	{attribute 'TcIecLibraryType'}
	{attribute 'external_name' := 'F_VN_ImageAbsoluteAverage_GUID_2A28D3C0_C84C_D0B6_A685_B52828B14CE3'}
	(* Computes the average absolute pixel value of an image. *)
	FUNCTION F_VN_ImageAbsoluteAverage : HRESULT
	VAR_INPUT
		ipSrcImage	:	ITcVnImage;	(* Source image *)
	END_VAR
	VAR_IN_OUT
		fAverage	:	LREAL;	(* Returns the average absolute pixel value *)
	END_VAR
	VAR_INPUT
		hrPrev	:	HRESULT;	(* HRESULT indicating the result of previous operations (If SUCCEEDED(hrPrev) equals false, no operation is executed.) *)
	END_VAR

END_FUNCTION

// Functions/Image Analysis/F_VN_ImageAverage

	{attribute 'TcIecLibraryType'}
	{attribute 'external_name' := 'F_VN_ImageAverage_GUID_FE774972_76AD_D27D_BAED_5933ADCB3F82'}
	(* Computes the (channel-wise) average pixel value of an image. *)
	FUNCTION F_VN_ImageAverage : HRESULT
	VAR_INPUT
		ipSrcImage	:	ITcVnImage;	(* Source image (1 - 4 channels) *)
	END_VAR
	VAR_IN_OUT
		aAverage	:	TcVnVector4_LREAL;	(* Returns the (channel-wise) average pixel value of ipSrcImage *)
	END_VAR
	VAR_INPUT
		hrPrev	:	HRESULT;	(* HRESULT indicating the result of previous operations (If SUCCEEDED(hrPrev) equals false, no operation is executed.) *)
	END_VAR

END_FUNCTION

// Functions/Image Analysis/F_VN_ImageAverageExp

	{attribute 'TcIecLibraryType'}
	{attribute 'external_name' := 'F_VN_ImageAverageExp_GUID_3E21A3C6_8FFA_DAD8_9B62_448D6BE9A6F9'}
	(* Computes the (channel-wise) average pixel value of an image. (expert function) *)
	FUNCTION F_VN_ImageAverageExp : HRESULT
	VAR_INPUT
		ipSrcImage	:	ITcVnImage;	(* Source image (1 - 4 channels) *)
	END_VAR
	VAR_IN_OUT
		aAverage	:	TcVnVector4_LREAL;	(* Returns the (channel-wise) average pixel value of ipSrcImage *)
	END_VAR
	VAR_INPUT
		ipMask	:	ITcVnImage;	(* Mask of type USINT (1 channel) *)
		hrPrev	:	HRESULT;	(* HRESULT indicating the result of previous operations (If SUCCEEDED(hrPrev) equals false, no operation is executed.) *)
	END_VAR

END_FUNCTION

// Functions/Image Analysis/F_VN_ImageAverageStdDev

	{attribute 'TcIecLibraryType'}
	{attribute 'external_name' := 'F_VN_ImageAverageStdDev_GUID_C9B349AB_3E58_D491_BF33_2DB560BD56B6'}
	(* Computes the (channel-wise) average pixel value and the corresponding standard deviation of an image. *)
	FUNCTION F_VN_ImageAverageStdDev : HRESULT
	VAR_INPUT
		ipSrcImage	:	ITcVnImage;	(* Source image (1 - 4 channels) *)
	END_VAR
	VAR_IN_OUT
		aAverage	:	TcVnVector4_LREAL;	(* Returns the (channel-wise) average pixel value of ipSrcImage *)
		aStdDev	:	TcVnVector4_LREAL;	(* Returns the (channel-wise) pixel value standard deviation of ipSrcImage *)
	END_VAR
	VAR_INPUT
		hrPrev	:	HRESULT;	(* HRESULT indicating the result of previous operations (If SUCCEEDED(hrPrev) equals false, no operation is executed.) *)
	END_VAR

END_FUNCTION

// Functions/Image Analysis/F_VN_ImageAverageStdDevExp

	{attribute 'TcIecLibraryType'}
	{attribute 'external_name' := 'F_VN_ImageAverageStdDevExp_GUID_869E8E6A_9652_D404_9B63_9DC2492C3981'}
	(* Computes the (channel-wise) average pixel value and the corresponding standard deviation of an image. (expert function) *)
	FUNCTION F_VN_ImageAverageStdDevExp : HRESULT
	VAR_INPUT
		ipSrcImage	:	ITcVnImage;	(* Source image (1 - 4 channels) *)
	END_VAR
	VAR_IN_OUT
		aAverage	:	TcVnVector4_LREAL;	(* Returns the (channel-wise) average pixel value of ipSrcImage *)
		aStdDev	:	TcVnVector4_LREAL;	(* Returns the (channel-wise) pixel value standard deviation of ipSrcImage *)
	END_VAR
	VAR_INPUT
		ipMask	:	ITcVnImage;	(* Mask of type USINT (1 channel) *)
		hrPrev	:	HRESULT;	(* HRESULT indicating the result of previous operations (If SUCCEEDED(hrPrev) equals false, no operation is executed.) *)
	END_VAR

END_FUNCTION

// Functions/Image Analysis/F_VN_ImageCenterOfMass

	{attribute 'TcIecLibraryType'}
	{attribute 'external_name' := 'F_VN_ImageCenterOfMass_GUID_E26AB96A_EBBA_D4BE_88C4_CC4D119BCFE3'}
	(* Computes the center of mass of an image. *)
	FUNCTION F_VN_ImageCenterOfMass : HRESULT
	VAR_INPUT
		ipSrcImage	:	ITcVnImage;	(* Source image (1 channel) *)
	END_VAR
	VAR_IN_OUT
		aCenterOfMass	:	TcVnPoint2_LREAL;	(* Returns the center of mass of the image *)
	END_VAR
	VAR_INPUT
		hrPrev	:	HRESULT;	(* HRESULT indicating the result of previous operations (If SUCCEEDED(hrPrev) equals false, no operation is executed.) *)
	END_VAR

END_FUNCTION

// Functions/Image Analysis/F_VN_ImageCenterOfMassExp

	{attribute 'TcIecLibraryType'}
	{attribute 'external_name' := 'F_VN_ImageCenterOfMassExp_GUID_59EB1D9F_B0E1_D491_9AD3_AE15A5EDCA0C'}
	(* Computes the center of mass of an image. *)
	FUNCTION F_VN_ImageCenterOfMassExp : HRESULT
	VAR_INPUT
		ipSrcImage	:	ITcVnImage;	(* Source image (1 channel) *)
	END_VAR
	VAR_IN_OUT
		aCenterOfMass	:	TcVnPoint2_LREAL;	(* Returns the center of mass of the image *)
	END_VAR
	VAR_INPUT
		ipMask	:	ITcVnImage;	(* Optional mask (1 channel of type USINT, same width and height as ipSrcImage) *)
		hrPrev	:	HRESULT;	(* HRESULT indicating the result of previous operations (If SUCCEEDED(hrPrev) equals false, no operation is executed.) *)
	END_VAR

END_FUNCTION

// Functions/Image Analysis/F_VN_ImageMedian

	{attribute 'TcIecLibraryType'}
	{attribute 'external_name' := 'F_VN_ImageMedian_GUID_F4FC4EAF_2294_D8BC_B4E8_1BD025C52AE2'}
	(* Computes the (approximated, channel-wise) median pixel value of an image. *)
	FUNCTION F_VN_ImageMedian : HRESULT
	VAR_INPUT
		ipSrcImage	:	ITcVnImage;	(* Source image (1 - 4 channels) *)
	END_VAR
	VAR_IN_OUT
		aMedian	:	TcVnVector4_LREAL;	(* Returns the (approximated, channel-wise) median pixel value of ipSrcImage *)
	END_VAR
	VAR_INPUT
		hrPrev	:	HRESULT;	(* HRESULT indicating the result of previous operations (If SUCCEEDED(hrPrev) equals false, no operation is executed.) *)
	END_VAR

END_FUNCTION

// Functions/Image Analysis/F_VN_ImageMedianExp

	{attribute 'TcIecLibraryType'}
	{attribute 'external_name' := 'F_VN_ImageMedianExp_GUID_743A193B_E592_DD8C_9D14_320E1F951A29'}
	(* Computes the (approximated, channel-wise) median pixel value of an image. (expert function) *)
	FUNCTION F_VN_ImageMedianExp : HRESULT
	VAR_INPUT
		ipSrcImage	:	ITcVnImage;	(* Source image (1 - 4 channels) *)
	END_VAR
	VAR_IN_OUT
		aMedian	:	TcVnVector4_LREAL;	(* Returns the (approximated, channel-wise) median pixel value of ipSrcImage *)
	END_VAR
	VAR_INPUT
		ipMask	:	ITcVnImage;	(* Mask of type USINT (1 channel) *)
		hrPrev	:	HRESULT;	(* HRESULT indicating the result of previous operations (If SUCCEEDED(hrPrev) equals false, no operation is executed.) *)
	END_VAR

END_FUNCTION

// Functions/Image Analysis/F_VN_ImageMoments

	{attribute 'TcIecLibraryType'}
	{attribute 'external_name' := 'F_VN_ImageMoments_GUID_E6E09E69_C28D_D19A_BF53_C7F25960A9B6'}
	(* Computes the spatial moments, the central moments, and the central normalized moments of an image up to the third order. *)
	FUNCTION F_VN_ImageMoments : HRESULT
	VAR_INPUT
		ipImage	:	ITcVnImage;	(* Source image (1 channel, elements of type USINT or REAL) *)
	END_VAR
	VAR_IN_OUT
		stMoments	:	TcVnMoments;	(* Returns a struct containing the moments *)
	END_VAR
	VAR_INPUT
		bBinaryImage	:	BOOL;	(* If true, all non-zero pixels are treated as ones *)
		hrPrev	:	HRESULT;	(* HRESULT indicating the result of previous operations (If SUCCEEDED(hrPrev) equals false, no operation is executed.) *)
	END_VAR

END_FUNCTION

// Functions/Image Analysis/F_VN_MaxPixelValue

	{attribute 'TcIecLibraryType'}
	{attribute 'external_name' := 'F_VN_MaxPixelValue_GUID_31A56A5D_0E05_D01A_8DEF_0E54450C3D06'}
	(* Finds the maximum pixel value in an image (1 - 4 channels supported). *)
	FUNCTION F_VN_MaxPixelValue : HRESULT
	VAR_INPUT
		ipImage	:	ITcVnImage;	(* Source image *)
	END_VAR
	VAR_IN_OUT
		aMaxValue	:	TcVnVector4_LREAL;	(* Returns the maximum pixel value *)
		aPosition	:	TcVnPoint2_DINT;	(* Returns the first found position of aMaxValue *)
	END_VAR
	VAR_INPUT
		hrPrev	:	HRESULT;	(* HRESULT indicating the result of previous operations (If SUCCEEDED(hrPrev) equals false, no operation is executed.) *)
	END_VAR

END_FUNCTION

// Functions/Image Analysis/F_VN_MaxPixelValueExp

	{attribute 'TcIecLibraryType'}
	{attribute 'external_name' := 'F_VN_MaxPixelValueExp_GUID_1D7E82B6_8AF8_D9FA_862F_06A78D41E2CB'}
	(* Finds the maximum pixel value in an image (1 - 4 channels supported). (expert function) *)
	FUNCTION F_VN_MaxPixelValueExp : HRESULT
	VAR_INPUT
		ipImage	:	ITcVnImage;	(* Source image *)
	END_VAR
	VAR_IN_OUT
		aMaxValue	:	TcVnVector4_LREAL;	(* Returns the maximum pixel value *)
		aPosition	:	TcVnPoint2_DINT;	(* Returns the first found position of aMaxValue (not supported for multi-channel images with ELEMENTWISE) *)
	END_VAR
	VAR_INPUT
		ipMask	:	ITcVnImage;	(* Optional mask to specify which pixel positions are considered (USINT, set parameter to 0 if not required) *)
		eVectorCompareMethod	:	ETcVnVectorCompareMethod;	(* Select a vector compare method for multi-channel images *)
		hrPrev	:	HRESULT;	(* HRESULT indicating the result of previous operations (If SUCCEEDED(hrPrev) equals false, no operation is executed.) *)
	END_VAR

END_FUNCTION

// Functions/Image Analysis/F_VN_MinPixelValue

	{attribute 'TcIecLibraryType'}
	{attribute 'external_name' := 'F_VN_MinPixelValue_GUID_5C49F054_DDB2_D937_AA1E_11C3D82EEE93'}
	(* Finds the minimum pixel value in an image (1 - 4 channels supported). *)
	FUNCTION F_VN_MinPixelValue : HRESULT
	VAR_INPUT
		ipImage	:	ITcVnImage;	(* Source image *)
	END_VAR
	VAR_IN_OUT
		aMinValue	:	TcVnVector4_LREAL;	(* Returns the minimum pixel value *)
		aPosition	:	TcVnPoint2_DINT;	(* Returns the first found position of aMinValue *)
	END_VAR
	VAR_INPUT
		hrPrev	:	HRESULT;	(* HRESULT indicating the result of previous operations (If SUCCEEDED(hrPrev) equals false, no operation is executed.) *)
	END_VAR

END_FUNCTION

// Functions/Image Analysis/F_VN_MinPixelValueExp

	{attribute 'TcIecLibraryType'}
	{attribute 'external_name' := 'F_VN_MinPixelValueExp_GUID_843B3B42_9C53_D824_9E8C_EE174779F5B7'}
	(* Finds the minimum pixel value in an image (1 - 4 channels supported). (expert function) *)
	FUNCTION F_VN_MinPixelValueExp : HRESULT
	VAR_INPUT
		ipImage	:	ITcVnImage;	(* Source image *)
	END_VAR
	VAR_IN_OUT
		aMinValue	:	TcVnVector4_LREAL;	(* Returns the minimum pixel value *)
		aPosition	:	TcVnPoint2_DINT;	(* Returns the first found position of aMinValue (not supported for multi-channel images with ELEMENTWISE) *)
	END_VAR
	VAR_INPUT
		ipMask	:	ITcVnImage;	(* Optional mask to specify which pixel positions are considered (USINT, set parameter to 0 if not required) *)
		eVectorCompareMethod	:	ETcVnVectorCompareMethod;	(* Select a vector compare method for multi-channel images *)
		hrPrev	:	HRESULT;	(* HRESULT indicating the result of previous operations (If SUCCEEDED(hrPrev) equals false, no operation is executed.) *)
	END_VAR

END_FUNCTION

// Functions/Image Analysis/F_VN_RegionOrientation

	{attribute 'TcIecLibraryType'}
	{attribute 'external_name' := 'F_VN_RegionOrientation_GUID_3030DDA5_1563_D8A7_A605_14FE25F90FB6'}
	(* Calculate the orientation of a region based on a binary image that contains a non zero value for every pixel in that region. *)
	FUNCTION F_VN_RegionOrientation : HRESULT
	VAR_INPUT
		ipSrcImage	:	ITcVnImage;	(* Source image (1 channel, binary). *)
	END_VAR
	VAR_IN_OUT
		stOrientation	:	TcVnRotatedRectangle;	(* Resulting rotated rectangle, containig center of mass, lenghts of axes, and rotation angle of the region in clockwise direction. *)
	END_VAR
	VAR_INPUT
		hrPrev	:	HRESULT;	(* HRESULT indicating the result of previous operations (If SUCCEEDED(hrPrev) equals false, no operation is executed.) *)
	END_VAR

END_FUNCTION

// Functions/Image Analysis/F_VN_RegionOrientationExp

	{attribute 'TcIecLibraryType'}
	{attribute 'external_name' := 'F_VN_RegionOrientationExp_GUID_2D852B8B_71E3_D6E2_B2E4_953101B92198'}
	(* Calculate the orientation of a region based on a binary image that contains a non zero value for every pixel in that region. (expert function) *)
	FUNCTION F_VN_RegionOrientationExp : HRESULT
	VAR_INPUT
		ipSrcImage	:	ITcVnImage;	(* Source image (1 channel, binary) *)
	END_VAR
	VAR_IN_OUT
		stOrientation	:	TcVnRotatedRectangle;	(* Resulting rotated rectangle, containig center of mass, lenghts of axes, and rotation angle of the region in clockwise direction. *)
	END_VAR
	VAR_INPUT
		eMethod	:	ETcVnOrientationMethod;	(* Method for calculating the orientation. *)
		hrPrev	:	HRESULT;	(* HRESULT indicating the result of previous operations (If SUCCEEDED(hrPrev) equals false, no operation is executed.) *)
	END_VAR

END_FUNCTION

// Functions/Image Analysis/F_VN_UprightInnerRectangle

	{attribute 'TcIecLibraryType'}
	{attribute 'external_name' := 'F_VN_UprightInnerRectangle_GUID_9A6E9260_7D1F_D847_92B8_836A9953FD1A'}
	(* Computes the maximum area upright inner rectangle inside an area. If the valid area contains very small invalid areas or the performance is too slow, use the expert variant of this function and manually choose a suitable nDownScaleFactor. *)
	FUNCTION F_VN_UprightInnerRectangle : HRESULT
	VAR_INPUT
		ipSrcImage	:	ITcVnImage;	(* Source image (USINT, 1 channel, binary, values > 0 mark valid area) *)
	END_VAR
	VAR_IN_OUT
		stRectangle	:	TcVnRectangle_DINT;	(* Returns the maximum area upright inner rectangle *)
	END_VAR
	VAR_INPUT
		hrPrev	:	HRESULT;	(* HRESULT indicating the result of previous operations (If SUCCEEDED(hrPrev) equals false, no operation is executed.) *)
	END_VAR

END_FUNCTION

// Functions/Image Analysis/F_VN_UprightInnerRectangleExp

	{attribute 'TcIecLibraryType'}
	{attribute 'external_name' := 'F_VN_UprightInnerRectangleExp_GUID_86F2F7A8_492B_D31B_B473_8128A9E0833D'}
	(* Computes the maximum area upright inner rectangle inside an area. (expert function) *)
	FUNCTION F_VN_UprightInnerRectangleExp : HRESULT
	VAR_INPUT
		ipSrcImage	:	ITcVnImage;	(* Source image (USINT, 1 channel, binary, values > 0 mark valid area) *)
	END_VAR
	VAR_IN_OUT
		stRectangle	:	TcVnRectangle_DINT;	(* Returns the maximum area upright inner rectangle *)
	END_VAR
	VAR_INPUT
		nDownScaleFactor	:	DINT;	(* To tradeoff performance vs. accuracy, a factor can be provided, to reduce the internally used image resolution. As long as invalid areas enclosed in the valid area are larger than nDownScaleFactor, the result usually still is the optimal one. Use -1 to auto select depending on ipSrcImage resolution, 0 to always use full resolution (slower but always optimal result). *)
		hrPrev	:	HRESULT;	(* HRESULT indicating the result of previous operations (If SUCCEEDED(hrPrev) equals false, no operation is executed.) *)
	END_VAR

END_FUNCTION

// Functions/Measurement/F_VN_AdjustSearchWindowOrientationToLinearEdge

	{attribute 'TcIecLibraryType'}
	{attribute 'external_name' := 'F_VN_AdjustSearchWindowOrientationToLinearEdge_GUID_D41518FD_A5A2_D4D6_B265_56FF46A599F0'}
	(* Adjust the search window to be orthogonal to a linear edge. Might be helpful before calling edge localization and distance measurement functions that rely on the search window. *)
	FUNCTION F_VN_AdjustSearchWindowOrientationToLinearEdge : HRESULT
	VAR_INPUT
		ipSrcImage	:	ITcVnImage;	(* Source image *)
	END_VAR
	VAR_IN_OUT
		aStartPoint	:	TcVnPoint2_REAL;	(* Position from which to start the search process (in the direction of aEndPoint), which is not changed *)
		aEndPoint	:	TcVnPoint2_REAL;	(* Position where the search process ends, which is adjusted by this function *)
	END_VAR
	VAR_INPUT
		eEdgeDirection	:	ETcVnEdgeDirection;	(* Specification of the edge direction to search for *)
		fMinStrength	:	REAL;	(* Specification of the minimum strength (intensity difference) of the edge to search for *)
		nMaxThickness	:	UDINT;	(* Specification of the maximum thickness of the edge to search for, which means fMinStrength must be reached within nMaxThickness pixels *)
		nSearchLines	:	UDINT;	(* Width of the search window, i.e. the number of search lines (3, 5, 7, ...), centered around the line specified by aStartPoint and aEndPoint *)
		hrPrev	:	HRESULT;	(* HRESULT indicating the result of previous operations (If SUCCEEDED(hrPrev) equals false, no operation is executed.) *)
	END_VAR

END_FUNCTION

// Functions/Measurement/F_VN_ClosestPointsBF

	{attribute 'TcIecLibraryType'}
	{attribute 'external_name' := 'F_VN_ClosestPointsBF_GUID_679941C9_C230_D8C5_8EC0_0DB38FAD54F3'}
	(* Find the closest distance between two 2d point sets of the same type, using a brute force approach. *)
	FUNCTION F_VN_ClosestPointsBF : HRESULT
	VAR_INPUT
		ipPointSet1	:	ITcVnContainer;	(* Container with 1st set of 2d points *)
		ipPointSet2	:	ITcVnContainer;	(* Container with 2nd set of 2d points *)
	END_VAR
	VAR_IN_OUT
		fMinDist	:	LREAL;	(* Returns the minimum distance between 2 points of the different point sets *)
		aPoint1	:	TcVnPoint2_LREAL;	(* Returns the point out of ipPointSet1, for which fMinDist is achieved *)
		aPoint2	:	TcVnPoint2_LREAL;	(* Returns the point out of ipPointSet2, for which fMinDist is achieved *)
	END_VAR
	VAR_INPUT
		hrPrev	:	HRESULT;	(* HRESULT indicating the result of previous operations (If SUCCEEDED(hrPrev) equals false, no operation is executed.) *)
	END_VAR

END_FUNCTION

// Functions/Measurement/F_VN_LocateCircularArc

	{attribute 'TcIecLibraryType'}
	{attribute 'external_name' := 'F_VN_LocateCircularArc_GUID_C374BA83_B360_D95C_BF1B_26CD74831828'}
	(* Locate a circular arc, using an interpolation method. *)
	FUNCTION F_VN_LocateCircularArc : HRESULT
	VAR_INPUT
		ipSrcImage	:	ITcVnImage;	(* Source image (1 channel) *)
	END_VAR
	VAR_IN_OUT
		stCircularArc	:	TcVnCircularArc;	(* Returns the circular arc parameters *)
		aCenter	:	TcVnPoint2_REAL;	(* Input estimated circle center (only used as a starting point to search for the circle contour, not used for the circle center estimation) *)
	END_VAR
	VAR_INPUT
		fSearchRadius	:	REAL;	(* Input search radius (starting from aCenter, should be greater than the actual circle radius but aCenter + fSearchRadius should be within the image borders) *)
		fArcDirectionRad	:	LREAL;	(* Input search starting direction in radian. Valid range is [-pi, +pi], where right is 0 rad, top is -pi/2 rad and bottom +pi/2 rad. The circular arc should at least be valid in range fArcDirectionRad +- 0.4 rad. *)
		eEdgeDirection	:	ETcVnEdgeDirection;	(* Specification of the edge direction to search for *)
		fMinStrength	:	REAL;	(* Specification of the minimum strength (intensity difference) of the edge to search for *)
		hrPrev	:	HRESULT;	(* HRESULT indicating the result of previous operations (If SUCCEEDED(hrPrev) equals false, no operation is executed.) *)
	END_VAR

END_FUNCTION

// Functions/Measurement/F_VN_LocateCircularArcExp

	{attribute 'TcIecLibraryType'}
	{attribute 'external_name' := 'F_VN_LocateCircularArcExp_GUID_4D7A20CA_FFD8_D52C_8A2B_7AF0F0C30851'}
	(* Locate a circular arc. (expert function) *)
	FUNCTION F_VN_LocateCircularArcExp : HRESULT
	VAR_INPUT
		ipSrcImage	:	ITcVnImage;	(* Source image (1 channel) *)
	END_VAR
	VAR_IN_OUT
		stCircularArc	:	TcVnCircularArc;	(* Returns the circular arc parameters *)
		aCenter	:	TcVnPoint2_REAL;	(* Input estimated circle center (only used as a starting point to search for the circle contour, not used for the circle center estimation) *)
	END_VAR
	VAR_INPUT
		fSearchRadius	:	REAL;	(* Input search radius (starting from aCenter, should be greater than the actual circle radius but aCenter + fSearchRadius should be within the image borders) *)
		fArcDirectionRad	:	LREAL;	(* Input search starting direction in radian. Valid range is [-pi, +pi], where right is 0 rad, top is -pi/2 rad and bottom +pi/2 rad. The circular arc should at least be valid in range fArcDirectionRad +- 4 * fAngleStepRad) *)
		eEdgeDirection	:	ETcVnEdgeDirection;	(* Specification of the edge direction to search for *)
		fMinStrength	:	REAL;	(* Specification of the minimum strength (intensity difference) of the edge to search for *)
		fAngleStepRad	:	LREAL;	(* Search step in rad (should be chosen so that about 20 - 60 steps are available for the whole arc. In most cases 0.1 rad (5.7 deg) is a good value) *)
		nMaxThickness	:	UDINT;	(* Specification of the maximum thickness of the edge to search for, which means fMinStrength must be reached within nMaxThickness pixels *)
		bInvertSearchDirection	:	BOOL;	(* If true, the search starts from outside the circular arc in direction of the center *)
		nSubpixelsIterations	:	UDINT;	(* Specifies the number of subpixels (for INTERPOLATION, 10 - 20 usually is sufficient) or maximum number of iterations for optimizing the parameters (for APPROX_ERF and APPROX_GAUSSIAN, 50 - 100 usually is sufficient) *)
		fApproxPrecision	:	REAL;	(* Specifies the approximation precision for APPROX_ERF and APPROX_GAUSSIAN (0.001 usually is sufficient, unused for INTERPOLATION) *)
		eAlgorithm	:	ETcVnEdgeDetectionAlgorithm;	(* Selection of the edge detection algorithm *)
		ipContourPoints	:	REFERENCE TO ITcVnContainer;	(* Returns the subpixel accurate contour (optional, set to 0 if not required; ContainerType_Vector_TcVnPoint2_REAL; Non-zero interface pointers are reused.) *)
		hrPrev	:	HRESULT;	(* HRESULT indicating the result of previous operations (If SUCCEEDED(hrPrev) equals false, no operation is executed.) *)
	END_VAR

END_FUNCTION

// Functions/Measurement/F_VN_LocateEdge

	{attribute 'TcIecLibraryType'}
	{attribute 'external_name' := 'F_VN_LocateEdge_GUID_F2889B56_A855_D692_90A0_C82CD37025D4'}
	(* Locate the points of the first occuring edge inside a specified search window, using an interpolation method. *)
	FUNCTION F_VN_LocateEdge : HRESULT
	VAR_INPUT
		ipSrcImage	:	ITcVnImage;	(* Source image (1 channel) *)
		ipEdgePoints	:	REFERENCE TO ITcVnContainer;	(* Returns the detected edge points (ContainerType_Vector_TcVnPoint2_REAL) *)
	END_VAR
	VAR_IN_OUT
		aStartPoint	:	TcVnPoint2_REAL;	(* Position from which to start the search process (in the direction of aEndPoint) *)
		aEndPoint	:	TcVnPoint2_REAL;	(* Position where the search process ends *)
	END_VAR
	VAR_INPUT
		eEdgeDirection	:	ETcVnEdgeDirection;	(* Specification of the edge direction to search for *)
		fMinStrength	:	REAL;	(* Specification of the minimum strength (intensity difference) of the edge to search for *)
		nSearchLines	:	UDINT;	(* Width of the search window, i.e. the number of search lines (1, 3, 5, 7, ...), centered around the line specified by aStartPoint and aEndPoint *)
		hrPrev	:	HRESULT;	(* HRESULT indicating the result of previous operations (If SUCCEEDED(hrPrev) equals false, no operation is executed.) *)
	END_VAR
	VAR_OUTPUT
		fAvgStrength	:	REAL;	(* Returns the average strength of the detected edge *)
	END_VAR

END_FUNCTION

// Functions/Measurement/F_VN_LocateEdgeExp

	{attribute 'TcIecLibraryType'}
	{attribute 'external_name' := 'F_VN_LocateEdgeExp_GUID_EE6B6E9D_DD5A_D666_A4B9_908FFEDDC4D1'}
	(* Locate the points of the first occuring edge inside a specified search window with subpixel accuracy. (expert function) *)
	FUNCTION F_VN_LocateEdgeExp : HRESULT
	VAR_INPUT
		ipSrcImage	:	ITcVnImage;	(* Source image (1 channel) *)
		ipEdgePoints	:	REFERENCE TO ITcVnContainer;	(* Returns the detected edge points (ContainerType_Vector_TcVnPoint2_REAL) *)
	END_VAR
	VAR_IN_OUT
		aStartPoint	:	TcVnPoint2_REAL;	(* Position from which to start the search process (in the direction of aEndPoint) *)
		aEndPoint	:	TcVnPoint2_REAL;	(* Position where the search process ends *)
	END_VAR
	VAR_INPUT
		eEdgeDirection	:	ETcVnEdgeDirection;	(* Specification of the edge direction to search for *)
		fMinStrength	:	REAL;	(* Specification of the minimum strength (intensity difference) of the edge to search for *)
		nSearchLines	:	UDINT;	(* Width of the search window, i.e. the number of search lines (1, 3, 5, 7, ...), centered around the line specified by aStartPoint and aEndPoint *)
		fSearchLineDist	:	REAL;	(* Distance between the search lines in pixels (> 0) *)
		nMaxThickness	:	UDINT;	(* Specification of the maximum thickness of the edge to search for, which means fMinStrength must be reached within nMaxThickness pixels *)
		nSubpixelsIterations	:	UDINT;	(* Specifies the number of subpixels (for INTERPOLATION, 10 - 20 usually is sufficient) or maximum number of iterations for optimizing the parameters (for APPROX_ERF and APPROX_GAUSSIAN, 50 - 100 usually is sufficient) *)
		fApproxPrecision	:	REAL;	(* Specifies the approximation precision for APPROX_ERF and APPROX_GAUSSIAN (0.001 usually is sufficient, unused for INTERPOLATION) *)
		eAlgorithm	:	ETcVnEdgeDetectionAlgorithm;	(* Selection of the edge detection algorithm *)
		hrPrev	:	HRESULT;	(* HRESULT indicating the result of previous operations (If SUCCEEDED(hrPrev) equals false, no operation is executed.) *)
	END_VAR
	VAR_OUTPUT
		fAvgStrength	:	REAL;	(* Returns the average strength of the detected edge *)
	END_VAR

END_FUNCTION

// Functions/Measurement/F_VN_LocateEdges

	{attribute 'TcIecLibraryType'}
	{attribute 'external_name' := 'F_VN_LocateEdges_GUID_89204EF8_C72B_D167_9AAC_2D5D7A2ADFBC'}
	(* Locate the points of multiple occuring edges inside a specified search window, using an interpolation method. *)
	FUNCTION F_VN_LocateEdges : HRESULT
	VAR_INPUT
		ipSrcImage	:	ITcVnImage;	(* Source image (1 channel) *)
		ipEdgePoints	:	REFERENCE TO ITcVnContainer;	(* Returns the detected edge points (ContainerType_Vector_Vector_TcVnPoint2_REAL) *)
	END_VAR
	VAR_IN_OUT
		aStartPoint	:	TcVnPoint2_REAL;	(* Position from which to start the search process (in the direction of aEndPoint) *)
		aEndPoint	:	TcVnPoint2_REAL;	(* Position where the search process ends *)
	END_VAR
	VAR_INPUT
		nNumEdges	:	UDINT;	(* The (maximum) number of edges to search for *)
		eEdgeDirection	:	ETcVnEdgeDirection;	(* Specification of the edge direction to search for *)
		bAlternateDirection	:	BOOL;	(* If true, eEdgeDirection is alternated after each detected edge. Else, only edges with eEdgeDirection are searched for. *)
		fMinStrength	:	REAL;	(* Specification of the minimum strength (intensity difference) of the edge to search for *)
		nSearchLines	:	UDINT;	(* Width of the search window, i.e. the number of search lines (1, 3, 5, 7, ...), centered around the line specified by aStartPoint and aEndPoint *)
		hrPrev	:	HRESULT;	(* HRESULT indicating the result of previous operations (If SUCCEEDED(hrPrev) equals false, no operation is executed.) *)
	END_VAR
	VAR_OUTPUT
		fAvgStrength	:	REAL;	(* Returns the average strength of the detected edges *)
	END_VAR

END_FUNCTION

// Functions/Measurement/F_VN_LocateEdgesExp

	{attribute 'TcIecLibraryType'}
	{attribute 'external_name' := 'F_VN_LocateEdgesExp_GUID_BB460134_7D54_D6AA_A05A_FB1C28B8BE51'}
	(* Locate the points of multiple occuring edges inside a specified search window with subpixel accuracy. (expert function) *)
	FUNCTION F_VN_LocateEdgesExp : HRESULT
	VAR_INPUT
		ipSrcImage	:	ITcVnImage;	(* Source image (1 channel) *)
		ipEdgePoints	:	REFERENCE TO ITcVnContainer;	(* Returns the detected edge points (ContainerType_Vector_Vector_TcVnPoint2_REAL) *)
	END_VAR
	VAR_IN_OUT
		aStartPoint	:	TcVnPoint2_REAL;	(* Position from which to start the search process (in the direction of aEndPoint) *)
		aEndPoint	:	TcVnPoint2_REAL;	(* Position where the search process ends *)
	END_VAR
	VAR_INPUT
		nNumEdges	:	UDINT;	(* The (maximum) number of edges to search for *)
		eEdgeDirection	:	ETcVnEdgeDirection;	(* Specification of the edge direction to search for *)
		bAlternateDirection	:	BOOL;	(* If true, eEdgeDirection is alternated after each detected edge. Else, only edges with eEdgeDirection are searched for. *)
		fMinStrength	:	REAL;	(* Specification of the minimum strength (intensity difference) of the edge to search for *)
		nSearchLines	:	UDINT;	(* Width of the search window, i.e. the number of search lines (1, 3, 5, 7, ...), centered around the line specified by aStartPoint and aEndPoint *)
		fSearchLineDist	:	REAL;	(* Distance between the search lines in pixels (> 0) *)
		nMaxThickness	:	UDINT;	(* Specification of the maximum thickness of the edge to search for, which means fMinStrength must be reached within nMaxThickness pixels *)
		nSubpixelsIterations	:	UDINT;	(* Specifies the number of subpixels (for INTERPOLATION, 10 - 20 usually is sufficient) or maximum number of iterations for optimizing the parameters (for APPROX_ERF and APPROX_GAUSSIAN, 50 - 100 usually is sufficient) *)
		fApproxPrecision	:	REAL;	(* Specifies the approximation precision for APPROX_ERF and APPROX_GAUSSIAN (0.001 usually is sufficient, unused for INTERPOLATION) *)
		eAlgorithm	:	ETcVnEdgeDetectionAlgorithm;	(* Selection of the edge detection algorithm *)
		hrPrev	:	HRESULT;	(* HRESULT indicating the result of previous operations (If SUCCEEDED(hrPrev) equals false, no operation is executed.) *)
	END_VAR
	VAR_OUTPUT
		fAvgStrength	:	REAL;	(* Returns the average strength of the detected edges *)
	END_VAR

END_FUNCTION

// Functions/Measurement/F_VN_LocateEllipse

	{attribute 'TcIecLibraryType'}
	{attribute 'external_name' := 'F_VN_LocateEllipse_GUID_E2BEEFE5_FDA4_D0A8_A984_F2C82F18D6F3'}
	(* Locate an ellipse, using an interpolation method for locating the edges. *)
	FUNCTION F_VN_LocateEllipse : HRESULT
	VAR_INPUT
		ipSrcImage	:	ITcVnImage;	(* Source image (1 channel) *)
	END_VAR
	VAR_IN_OUT
		stEllipse	:	TcVnRotatedRectangle;	(* Returns the detected ellipse *)
		aCenter	:	TcVnPoint2_REAL;	(* The expected ellipse center *)
	END_VAR
	VAR_INPUT
		fSearchRadius	:	REAL;	(* Radius around aCenter to search for edges (aCenter + fSearchRadius in all directions must be inside image borders!) *)
		eEdgeDirection	:	ETcVnEdgeDirection;	(* Specification of the edge direction to search for (from center to outside ellipse) *)
		fMinStrength	:	REAL;	(* Specification of the minimum strength (intensity difference) of the edge to search for *)
		hrPrev	:	HRESULT;	(* HRESULT indicating the result of previous operations (If SUCCEEDED(hrPrev) equals false, no operation is executed.) *)
	END_VAR

END_FUNCTION

// Functions/Measurement/F_VN_LocateEllipseExp

	{attribute 'TcIecLibraryType'}
	{attribute 'external_name' := 'F_VN_LocateEllipseExp_GUID_958DA967_81A5_DFC3_B424_5FAC80BB3AA0'}
	(* Locate an ellipse. (expert function) *)
	FUNCTION F_VN_LocateEllipseExp : HRESULT
	VAR_INPUT
		ipSrcImage	:	ITcVnImage;	(* Source image (1 channel) *)
	END_VAR
	VAR_IN_OUT
		stEllipse	:	TcVnRotatedRectangle;	(* Returns the detected ellipse *)
		aCenter	:	TcVnPoint2_REAL;	(* The expected ellipse center *)
	END_VAR
	VAR_INPUT
		fSearchRadius	:	REAL;	(* Radius around aCenter to search for edges *)
		eEdgeDirection	:	ETcVnEdgeDirection;	(* Specification of the edge direction to search for (from center to outside ellipse or other way round, if bInvertSearchDirection is true) *)
		fMinStrength	:	REAL;	(* Specification of the minimum strength (intensity difference) of the edge to search for *)
		nMaxThickness	:	UDINT;	(* Specification of the maximum thickness of the edge to search for, which means fMinStrength must be reached within nMaxThickness pixels *)
		bInvertSearchDirection	:	BOOL;	(* If true, the search starts from outside the ellipse in direction of the center *)
		fMinSearchRadius	:	REAL;	(* Radius around aCenter to skip before starting to search for edges (e.g. to save time or if the center contains edges that should be ignored) *)
		nSubpixelsIterations	:	UDINT;	(* Specifies the number of subpixels (for INTERPOLATION, 10 - 20 usually is sufficient) or maximum number of iterations for optimizing the parameters (for APPROX_ERF and APPROX_GAUSSIAN, 50 - 100 usually is sufficient) *)
		nSearchLines	:	UDINT;	(* Specifies the amount of search lines, which are equally distributed in all directions (must be >= 8 and a multiple of 4) *)
		fApproxPrecision	:	REAL;	(* Specifies the approximation precision for APPROX_ERF and APPROX_GAUSSIAN (0.001 usually is sufficient, unused for INTERPOLATION) *)
		eAlgorithm	:	ETcVnEdgeDetectionAlgorithm;	(* Selection of the edge detection algorithm *)
		ipContourPoints	:	REFERENCE TO ITcVnContainer;	(* Returns the subpixel accurate ellipse contour (optional, set to 0 if not required; ContainerType_Vector_TcVnPoint2_REAL; Non-zero interface pointers are reused.) *)
		hrPrev	:	HRESULT;	(* HRESULT indicating the result of previous operations (If SUCCEEDED(hrPrev) equals false, no operation is executed.) *)
	END_VAR

END_FUNCTION

// Functions/Measurement/F_VN_MeasureAngleBetweenEdges

	{attribute 'TcIecLibraryType'}
	{attribute 'external_name' := 'F_VN_MeasureAngleBetweenEdges_GUID_4FA8BC1E_0BCD_DC7A_B904_883E49E6A3D8'}
	(* Measure the angle between 2 edges, using an interpolation method. *)
	FUNCTION F_VN_MeasureAngleBetweenEdges : HRESULT
	VAR_INPUT
		ipSrcImage	:	ITcVnImage;	(* Source image (1 channel) *)
	END_VAR
	VAR_IN_OUT
		fAngle	:	REAL;	(* Returns the angle between the detected edges (radians) *)
		aInnerPoint	:	TcVnPoint2_REAL;	(* Position inside the angle to measure, from which to start the edge search process (in the direction of aOuterPoint1 and aOuterPoint2) *)
		aOuterPoint1	:	TcVnPoint2_REAL;	(* Position where the search process for edge 1 ends *)
		aOuterPoint2	:	TcVnPoint2_REAL;	(* Position where the search process for edge 2 ends *)
	END_VAR
	VAR_INPUT
		eEdgeDirection	:	ETcVnEdgeDirection;	(* Specification of the edge direction from aInnerPoint to aOuterPoint1 and aOuterPoint2 to search for *)
		fMinStrength	:	REAL;	(* Specification of the minimum strength (intensity difference) of the edge to search for *)
		nSearchLines	:	UDINT;	(* Width of the search windows, i.e. the number of search lines (3, 5, 7, ...), centered around the lines specified by aInnerPoint and aOuterPoint1, aOuterPoint2 *)
		hrPrev	:	HRESULT;	(* HRESULT indicating the result of previous operations (If SUCCEEDED(hrPrev) equals false, no operation is executed.) *)
	END_VAR

END_FUNCTION

// Functions/Measurement/F_VN_MeasureAngleBetweenEdgesExp

	{attribute 'TcIecLibraryType'}
	{attribute 'external_name' := 'F_VN_MeasureAngleBetweenEdgesExp_GUID_261197EF_E520_DF25_8F1E_4CADE9E87269'}
	(* Measure the angle between 2 edges. *)
	FUNCTION F_VN_MeasureAngleBetweenEdgesExp : HRESULT
	VAR_INPUT
		ipSrcImage	:	ITcVnImage;	(* Source image (1 channel) *)
	END_VAR
	VAR_IN_OUT
		fAngle	:	REAL;	(* Returns the angle between the detected edges (radians or degrees, depending on bAngleInDegrees) *)
		aInnerPoint	:	TcVnPoint2_REAL;	(* Position inside the angle to measure, from which to start the edge search process (in the direction of aOuterPoint1 and aOuterPoint2) *)
		aOuterPoint1	:	TcVnPoint2_REAL;	(* Position where the search process for edge 1 ends *)
		aOuterPoint2	:	TcVnPoint2_REAL;	(* Position where the search process for edge 2 ends *)
	END_VAR
	VAR_INPUT
		eEdgeDirection	:	ETcVnEdgeDirection;	(* Specification of the edge direction from aInnerPoint to aOuterPoint1 and aOuterPoint2 to search for *)
		fMinStrength	:	REAL;	(* Specification of the minimum strength (intensity difference) of the edge to search for *)
		nSearchLines	:	UDINT;	(* Width of the search window, i.e. the number of search lines (3, 5, 7, ...), centered around the line specified by aInnerPoint and aOuterPoint1, aOuterPoint2 *)
		fSearchLineDist	:	REAL;	(* Distance between the search lines in pixels (> 0) *)
		nMaxThickness	:	UDINT;	(* Specification of the maximum thickness of the edge to search for, which means fMinStrength must be reached within nMaxThickness pixels *)
		bInvertSearchDirection	:	BOOL;	(* If true, the search starts from each aOuterPoint in direction of aInnerPoint *)
		nSubpixelsIterations	:	UDINT;	(* Specifies the number of subpixels (for INTERPOLATION, 10 - 20 usually is sufficient) or maximum number of iterations for optimizing the parameters (for APPROX_ERF and APPROX_GAUSSIAN, 50 - 100 usually is sufficient) *)
		bAngleInDegrees	:	BOOL;	(* fAngle is in degrees, if true *)
		fApproxPrecision	:	REAL;	(* Specifies the approximation precision for APPROX_ERF and APPROX_GAUSSIAN (0.001 usually is sufficient, unused for INTERPOLATION) *)
		eAlgorithm	:	ETcVnEdgeDetectionAlgorithm;	(* Selection of the edge detection algorithm *)
		ipEdgePoints1	:	REFERENCE TO ITcVnContainer;	(* Returns the detected edge points between aInnerPoint and aOuterPoint1 (ContainerType_Vector_TcVnPoint2_REAL) *)
		ipEdgePoints2	:	REFERENCE TO ITcVnContainer;	(* Returns the detected edge points between aInnerPoint and aOuterPoint2 (ContainerType_Vector_TcVnPoint2_REAL) *)
		hrPrev	:	HRESULT;	(* HRESULT indicating the result of previous operations (If SUCCEEDED(hrPrev) equals false, no operation is executed.) *)
	END_VAR

END_FUNCTION

// Functions/Measurement/F_VN_MeasureEdgeDistance

	{attribute 'TcIecLibraryType'}
	{attribute 'external_name' := 'F_VN_MeasureEdgeDistance_GUID_F4DC5D30_AF71_D56D_B2C6_0402FE47CEED'}
	(* Measure the distance between 2 parallel edges, using an interpolation method. *)
	FUNCTION F_VN_MeasureEdgeDistance : HRESULT
	VAR_INPUT
		ipSrcImage	:	ITcVnImage;	(* Source image (1 channel) *)
	END_VAR
	VAR_IN_OUT
		fAvgDistance	:	REAL;	(* Returns the average distance between the detected edges *)
		aStartPoint	:	TcVnPoint2_REAL;	(* Position from which to start the search process (in the direction of aEndPoint) *)
		aEndPoint	:	TcVnPoint2_REAL;	(* Position where the search process ends *)
	END_VAR
	VAR_INPUT
		eEdgeDirection	:	ETcVnEdgeDirection;	(* Specification of the edge direction from aStartPoint to aEndPoint to search for *)
		fMinStrength	:	REAL;	(* Specification of the minimum strength (intensity difference) of the edge to search for *)
		nSearchLines	:	UDINT;	(* Width of the search window, i.e. the number of search lines (1, 3, 5, 7, ...), centered around the line specified by aStartPoint and aEndPoint *)
		hrPrev	:	HRESULT;	(* HRESULT indicating the result of previous operations (If SUCCEEDED(hrPrev) equals false, no operation is executed.) *)
	END_VAR

END_FUNCTION

// Functions/Measurement/F_VN_MeasureEdgeDistanceExp

	{attribute 'TcIecLibraryType'}
	{attribute 'external_name' := 'F_VN_MeasureEdgeDistanceExp_GUID_2A4B8E0A_21E6_DBC7_BEF7_445F09C31B54'}
	(* Measure the distance between 2 parallel edges. (expert function) *)
	FUNCTION F_VN_MeasureEdgeDistanceExp : HRESULT
	VAR_INPUT
		ipSrcImage	:	ITcVnImage;	(* Source image (1 channel) *)
	END_VAR
	VAR_IN_OUT
		fAvgDistance	:	REAL;	(* Returns the average distance between the detected edges *)
		aStartPoint	:	TcVnPoint2_REAL;	(* Position from which to start the search process (in the direction of aEndPoint) *)
		aEndPoint	:	TcVnPoint2_REAL;	(* Position where the search process ends *)
	END_VAR
	VAR_INPUT
		eEdgeDirection	:	ETcVnEdgeDirection;	(* Specification of the edge direction from aStartPoint to aEndPoint to search for *)
		fMinStrength	:	REAL;	(* Specification of the minimum strength (intensity difference) of the edge to search for *)
		nSearchLines	:	UDINT;	(* Width of the search window, i.e. the number of search lines (1, 3, 5, 7, ...), centered around the line specified by aStartPoint and aEndPoint *)
		fSearchLineDist	:	REAL;	(* Distance between the search lines in pixels (> 0) *)
		nMaxThickness	:	UDINT;	(* Specification of the maximum thickness of the edge to search for, which means fMinStrength must be reached within nMaxThickness pixels *)
		bInvertSearchDirection	:	BOOL;	(* If true, the search starts from the center point between aStartPoint and aEndPoint in both directions *)
		fSearchGap	:	REAL;	(* Optional width of a gap (>= 0, centered between aStartPoint and aEndPoint), that is neglected for searching edges (can reduce execution time). The 2 edges to search for must be on different sides of the gap. *)
		nSubpixelsIterations	:	UDINT;	(* Specifies the number of subpixels (for INTERPOLATION, 10 - 20 usually is sufficient) or maximum number of iterations for optimizing the parameters (for APPROX_ERF and APPROX_GAUSSIAN, 50 - 100 usually is sufficient) *)
		fApproxPrecision	:	REAL;	(* Specifies the approximation precision for APPROX_ERF and APPROX_GAUSSIAN (0.001 usually is sufficient, unused for INTERPOLATION) *)
		eAlgorithm	:	ETcVnEdgeDetectionAlgorithm;	(* Selection of the edge detection algorithm *)
		ipEdgePoints1	:	REFERENCE TO ITcVnContainer;	(* Returns the detected edge points of the edge near aStartPoint (optional, set to 0 if not required; ContainerType_Vector_TcVnPoint2_REAL) *)
		ipEdgePoints2	:	REFERENCE TO ITcVnContainer;	(* Returns the detected edge points of the edge near aEndPoint (optional, set to 0 if not required; ContainerType_Vector_TcVnPoint2_REAL) *)
		ipDistances	:	REFERENCE TO ITcVnContainer;	(* Returns the distances between the detected edge points (optional, set to 0 if not required; ContainerType_Vector_REAL) *)
		hrPrev	:	HRESULT;	(* HRESULT indicating the result of previous operations (If SUCCEEDED(hrPrev) equals false, no operation is executed.) *)
	END_VAR

END_FUNCTION

// Functions/Measurement/F_VN_MeasureMinEdgeDistance

	{attribute 'TcIecLibraryType'}
	{attribute 'external_name' := 'F_VN_MeasureMinEdgeDistance_GUID_32880315_7CC1_DF1F_BA90_990C32E9EC6C'}
	(* Measure the minimum distance within the specified search window between 2 edges, using an interpolation method. *)
	FUNCTION F_VN_MeasureMinEdgeDistance : HRESULT
	VAR_INPUT
		ipSrcImage	:	ITcVnImage;	(* Source image (1 channel) *)
	END_VAR
	VAR_IN_OUT
		fMinDistance	:	REAL;	(* Returns the minimum distance between the detected edges *)
		aStartPoint	:	TcVnPoint2_REAL;	(* Position from which to start the search process (in the direction of aEndPoint) *)
		aEndPoint	:	TcVnPoint2_REAL;	(* Position where the search process ends *)
	END_VAR
	VAR_INPUT
		eEdgeDirection	:	ETcVnEdgeDirection;	(* Specification of the edge direction from aStartPoint to aEndPoint to search for *)
		fMinStrength	:	REAL;	(* Specification of the minimum strength (intensity difference) of the edge to search for *)
		nSearchLines	:	UDINT;	(* Width of the search window, i.e. the number of search lines (1, 3, 5, 7, ...), centered around the line specified by aStartPoint and aEndPoint *)
		hrPrev	:	HRESULT;	(* HRESULT indicating the result of previous operations (If SUCCEEDED(hrPrev) equals false, no operation is executed.) *)
	END_VAR

END_FUNCTION

// Functions/Measurement/F_VN_MeasureMinEdgeDistanceExp

	{attribute 'TcIecLibraryType'}
	{attribute 'external_name' := 'F_VN_MeasureMinEdgeDistanceExp_GUID_8425933C_5E0C_D8D9_B48D_2A6F0C488F9B'}
	(* Measure the minimum distance within the specified search window between 2 edges. (expert function) *)
	FUNCTION F_VN_MeasureMinEdgeDistanceExp : HRESULT
	VAR_INPUT
		ipSrcImage	:	ITcVnImage;	(* Source image (1 channel) *)
	END_VAR
	VAR_IN_OUT
		fMinDistance	:	REAL;	(* Returns the minimum distance between the detected edges *)
		aStartPoint	:	TcVnPoint2_REAL;	(* Position from which to start the search process (in the direction of aEndPoint) *)
		aEndPoint	:	TcVnPoint2_REAL;	(* Position where the search process ends *)
	END_VAR
	VAR_INPUT
		eEdgeDirection	:	ETcVnEdgeDirection;	(* Specification of the edge direction from aStartPoint to aEndPoint to search for *)
		fMinStrength	:	REAL;	(* Specification of the minimum strength (intensity difference) of the edge to search for *)
		nSearchLines	:	UDINT;	(* Width of the search window, i.e. the number of search lines (1, 3, 5, 7, ...), centered around the line specified by aStartPoint and aEndPoint *)
		fSearchLineDist	:	REAL;	(* Distance between the search lines in pixels (> 0) *)
		nMaxThickness	:	UDINT;	(* Specification of the maximum thickness of the edge to search for, which means fMinStrength must be reached within nMaxThickness pixels *)
		bInvertSearchDirection	:	BOOL;	(* If true, the search starts from the center point between aStartPoint and aEndPoint in both directions *)
		fSearchGap	:	REAL;	(* Optional width of a gap (>= 0, centered between aStartPoint and aEndPoint), that is neglected for searching edges (can reduce execution time). The 2 edges to search for must be on different sides of the gap. *)
		nSubpixelsIterations	:	UDINT;	(* Specifies the number of subpixels (for INTERPOLATION, 10 - 20 usually is sufficient) or maximum number of iterations for optimizing the parameters (for APPROX_ERF and APPROX_GAUSSIAN, 50 - 100 usually is sufficient) *)
		fApproxPrecision	:	REAL;	(* Specifies the approximation precision for APPROX_ERF and APPROX_GAUSSIAN (0.001 usually is sufficient, unused for INTERPOLATION) *)
		eAlgorithm	:	ETcVnEdgeDetectionAlgorithm;	(* Selection of the edge detection algorithm *)
		ipEdgePoints1	:	REFERENCE TO ITcVnContainer;	(* Returns the detected edge points of the edge near aStartPoint (optional, set to 0 if not required; ContainerType_Vector_TcVnPoint2_REAL) *)
		ipEdgePoints2	:	REFERENCE TO ITcVnContainer;	(* Returns the detected edge points of the edge near aEndPoint (optional, set to 0 if not required; ContainerType_Vector_TcVnPoint2_REAL) *)
	END_VAR
	VAR_IN_OUT
		aPoint1	:	TcVnPoint2_REAL;	(* Returns the point on the edge near aStartPoint, for which the minimum distance is achieved *)
		aPoint2	:	TcVnPoint2_REAL;	(* Returns the point on the edge near aEndPoint, for which the minimum distance is achieved *)
	END_VAR
	VAR_INPUT
		hrPrev	:	HRESULT;	(* HRESULT indicating the result of previous operations (If SUCCEEDED(hrPrev) equals false, no operation is executed.) *)
	END_VAR

END_FUNCTION

// Functions/Basic Container Operations/F_VN_AdvanceIterator

	{attribute 'TcIecLibraryType'}
	{attribute 'external_name' := 'F_VN_AdvanceIterator_GUID_24AA54BD_71F7_D985_8DE7_BCFAB184EA09'}
	(* Advance an iterator by the specified offset. *)
	FUNCTION F_VN_AdvanceIterator : HRESULT
	VAR_INPUT
		ipIterator	:	ITcVnForwardIterator;	(* Iterator to be advanced *)
		nOffset	:	LINT;	(* Offset, by which ipIterator is advanced *)
		hrPrev	:	HRESULT;	(* HRESULT indicating the result of previous operations (If SUCCEEDED(hrPrev) equals false, no operation is executed.) *)
	END_VAR

END_FUNCTION

// Functions/Basic Container Operations/F_VN_CheckIfEmpty

	{attribute 'TcIecLibraryType'}
	{attribute 'external_name' := 'F_VN_CheckIfEmpty_GUID_7F482D8D_1CA5_D20C_B8C3_97B1F169FECB'}
	(* Checks if the container is empty. (Alternatively use interface method .CheckIfEmpty.) *)
	FUNCTION F_VN_CheckIfEmpty : HRESULT
	VAR_INPUT
		ipContainer	:	ITcVnContainer;	(* Container *)
		hrPrev	:	HRESULT;	(* HRESULT indicating the result of previous operations (If SUCCEEDED(hrPrev) equals false, no operation is executed.) *)
	END_VAR

END_FUNCTION

// Functions/Basic Container Operations/F_VN_CheckIfIteratorIsAtEnd

	{attribute 'TcIecLibraryType'}
	{attribute 'external_name' := 'F_VN_CheckIfIteratorIsAtEnd_GUID_B8A07D30_99DC_D2BF_A34B_16C21C8D6288'}
	(* Checks if the iterator points to the past-the-end element. (Alternatively use interface method .CheckIfEnd.) *)
	FUNCTION F_VN_CheckIfIteratorIsAtEnd : HRESULT
	VAR_INPUT
		ipIterator	:	ITcVnForwardIterator;	(* Iterator *)
		hrPrev	:	HRESULT;	(* HRESULT indicating the result of previous operations (If SUCCEEDED(hrPrev) equals false, no operation is executed.) *)
	END_VAR

END_FUNCTION

// Functions/Basic Container Operations/F_VN_ConvertContainerType

	{attribute 'TcIecLibraryType'}
	{attribute 'external_name' := 'F_VN_ConvertContainerType_GUID_89C340AA_711E_D555_89CC_2BC6819B1313'}
	(* Converts a container to another type (Struct element types are not supported). *)
	FUNCTION F_VN_ConvertContainerType : HRESULT
	VAR_INPUT
		ipSrcContainer	:	ITcVnContainer;	(* Source container *)
		ipDestContainer	:	REFERENCE TO ITcVnContainer;	(* Returns the converted container *)
		nDestTypeGuid	:	GUID;	(* Specifies the destination container type for the conversion *)
		hrPrev	:	HRESULT;	(* HRESULT indicating the result of previous operations (If SUCCEEDED(hrPrev) equals false, no operation is executed.) *)
	END_VAR

END_FUNCTION

// Functions/Basic Container Operations/F_VN_CopyContainer

	{attribute 'TcIecLibraryType'}
	{attribute 'external_name' := 'F_VN_CopyContainer_GUID_52C11E05_B7B0_D697_9758_9B5F18270AF8'}
	(* Copys a container. *)
	FUNCTION F_VN_CopyContainer : HRESULT
	VAR_INPUT
		ipSrcContainer	:	ITcVnContainer;	(* Source container *)
		ipDestContainer	:	REFERENCE TO ITcVnContainer;	(* Destination container (same type ID as ipSrcContainer; Non-zero interface pointers are reused.) *)
		hrPrev	:	HRESULT;	(* HRESULT indicating the result of previous operations (If SUCCEEDED(hrPrev) equals false, no operation is executed.) *)
	END_VAR

END_FUNCTION

// Functions/Basic Container Operations/F_VN_CopyContainerElementsConditional_ITcVnContainer

	{attribute 'TcIecLibraryType'}
	{attribute 'external_name' := 'F_VN_CopyContainerElementsConditional_ITcVnContainer_GUID_A724F0D8_9B12_D670_A6EC_1BC75E575586'}
	(* Copys container elements to a new container, depending on a custom condition. *)
	FUNCTION F_VN_CopyContainerElementsConditional_ITcVnContainer : HRESULT
	VAR_INPUT
		ipSrcContainer	:	ITcVnContainer;	(* Source container *)
		ipDestContainer	:	REFERENCE TO ITcVnContainer;	(* Returns a container with elements, that match the condition *)
		ipConditionFB	:	ITcVnCustomElementCondition_ITcVnContainer;	(* Custom condition *)
		hrPrev	:	HRESULT;	(* HRESULT indicating the result of previous operations (If SUCCEEDED(hrPrev) equals false, no operation is executed.) *)
	END_VAR

END_FUNCTION

// Interfaces/Containers/Function Blocks/ITcVnCustomElementCondition_ITcVnContainer

	(* Offers an interface for a custom condition computed for a container. *)
	{attribute 'c++_compatible'}
	INTERFACE ITcVnCustomElementCondition_ITcVnContainer


(* Evaluates the condition for the container. *)
	{attribute 'c++_compatible'}
	{attribute 'minimal_input_size' := '4'}
	{attribute 'pack_mode' := '4'}
	METHOD Condition : BOOL
	VAR_INPUT
		ipElement : ITcVnContainer;
	END_VAR
END_METHOD

END_INTERFACE

// Functions/Basic Container Operations/F_VN_CopyContainerElementsConditional_ITcVnForwardIterator

	{attribute 'TcIecLibraryType'}
	{attribute 'external_name' := 'F_VN_CopyContainerElementsConditional_ITcVnForwardIterator_GUID_CB3EABC9_4F32_D01D_A1E5_F8CD523522AE'}
	(* Copys container elements to a new container, depending on a custom condition. *)
	FUNCTION F_VN_CopyContainerElementsConditional_ITcVnForwardIterator : HRESULT
	VAR_INPUT
		ipSrcContainer	:	ITcVnContainer;	(* Source container *)
		ipDestContainer	:	REFERENCE TO ITcVnContainer;	(* Returns a container with elements, that match the condition *)
		ipConditionFB	:	ITcVnCustomElementCondition_ITcVnForwardIterator;	(* Custom condition *)
		hrPrev	:	HRESULT;	(* HRESULT indicating the result of previous operations (If SUCCEEDED(hrPrev) equals false, no operation is executed.) *)
	END_VAR

END_FUNCTION

// Interfaces/Containers/Function Blocks/ITcVnCustomElementCondition_ITcVnForwardIterator

	(* Offers an interface for a custom condition computed for an element represented by an ITcVnForwardIterator. *)
	{attribute 'c++_compatible'}
	INTERFACE ITcVnCustomElementCondition_ITcVnForwardIterator


(* Evaluates the condition for the provided element. *)
	{attribute 'c++_compatible'}
	{attribute 'minimal_input_size' := '4'}
	{attribute 'pack_mode' := '4'}
	METHOD Condition : BOOL
	VAR_INPUT
		ipElement : ITcVnForwardIterator;
	END_VAR
END_METHOD

END_INTERFACE

// Functions/Basic Container Operations/F_VN_CreateContainer

	{attribute 'TcIecLibraryType'}
	{attribute 'external_name' := 'F_VN_CreateContainer_GUID_E9B1C4D3_2307_D2FA_BB55_905A760F0DDB'}
	(* Creates a container with type GUID nTypeGuid and return its container interface. *)
	FUNCTION F_VN_CreateContainer : HRESULT
	VAR_INPUT
		ipContainer	:	REFERENCE TO ITcVnContainer;	(* Returns the created container *)
		nTypeGuid	:	GUID;	(* Type GUID of the container to be created *)
		nElementNum	:	ULINT;	(* Number of elements *)
		hrPrev	:	HRESULT;	(* HRESULT indicating the result of previous operations (If SUCCEEDED(hrPrev) equals false, no operation is executed.) *)
	END_VAR

END_FUNCTION

// Functions/Basic Container Operations/F_VN_CreateContainerFromArray

	{attribute 'TcIecLibraryType'}
	{attribute 'external_name' := 'F_VN_CreateContainerFromArray_GUID_2239801F_E9BB_DE0B_9285_690EA2BC071A'}
	(* Creates a container with type GUID nTypeGuid, initialize it with provided data and return its container interface. Only supported for basic container types, i.e. not for containers of containers. *)
	FUNCTION F_VN_CreateContainerFromArray : HRESULT
	VAR_INPUT
		pData	:	PVOID;	(* Pointer to the data array. Make sure that the array contains at least nElementNum elements and that the array element type matches the container element type. *)
		ipContainer	:	REFERENCE TO ITcVnContainer;	(* Returns the created container *)
		nTypeGuid	:	GUID;	(* Type GUID of the container to be created *)
		nElementNum	:	ULINT;	(* Number of elements to copy from pData *)
		hrPrev	:	HRESULT;	(* HRESULT indicating the result of previous operations (If SUCCEEDED(hrPrev) equals false, no operation is executed.) *)
	END_VAR

END_FUNCTION

// Functions/Basic Container Operations/F_VN_EraseFromContainer

	{attribute 'TcIecLibraryType'}
	{attribute 'external_name' := 'F_VN_EraseFromContainer_GUID_5EE4FFDB_E77D_DDBD_B0FB_7BFB996E54F2'}
	(* Erase elements from a container. *)
	FUNCTION F_VN_EraseFromContainer : HRESULT
	VAR_INPUT
		ipContainer	:	ITcVnContainer;	(* Container from which to erase elements *)
		nStartIdx	:	ULINT;	(* Index of the first element to erase *)
		nCount	:	ULINT;	(* Number of elements to erase *)
		hrPrev	:	HRESULT;	(* HRESULT indicating the result of previous operations (If SUCCEEDED(hrPrev) equals false, no operation is executed.) *)
	END_VAR

END_FUNCTION

// Functions/Basic Container Operations/F_VN_ExportContainer

	{attribute 'TcIecLibraryType'}
	{attribute 'external_name' := 'F_VN_ExportContainer_GUID_3B72E028_7190_DC74_86E0_D3C8698A322A'}
	(* Export the container elements into a buffer (e.g. an array). Only possible for containers with basic elements. *)
	FUNCTION F_VN_ExportContainer : HRESULT
	VAR_INPUT
		ipContainer	:	ITcVnContainer;	(* Container with basic elements *)
		pBuffer	:	PVOID;	(* Buffer to store the container elements (Make sure to allocate enough memory! The required size in bytes can be determined using the function F_VN_ExportContainerSize) *)
		nBufferSize	:	ULINT;	(* Size of the buffer memory in bytes *)
		hrPrev	:	HRESULT;	(* HRESULT indicating the result of previous operations (If SUCCEEDED(hrPrev) equals false, no operation is executed.) *)
	END_VAR

END_FUNCTION

// Functions/Basic Container Operations/F_VN_ExportContainerSize

	{attribute 'TcIecLibraryType'}
	{attribute 'external_name' := 'F_VN_ExportContainerSize_GUID_FE960675_53CE_D337_8BE0_1063D1BD3F6A'}
	(* Determine the required buffer size in bytes to store all container elements (number_of_Elements * size_per_Element). Only possible for containers with basic elements. *)
	FUNCTION F_VN_ExportContainerSize : HRESULT
	VAR_INPUT
		ipContainer	:	ITcVnContainer;	(* Container with basic elements *)
	END_VAR
	VAR_IN_OUT
		nBufferSize	:	ULINT;	(* Output parameter containing the required buffer size *)
	END_VAR
	VAR_INPUT
		hrPrev	:	HRESULT;	(* HRESULT indicating the result of previous operations (If SUCCEEDED(hrPrev) equals false, no operation is executed.) *)
	END_VAR

END_FUNCTION

// Functions/Basic Container Operations/F_VN_ExportContainer_String

	{attribute 'TcIecLibraryType'}
	{attribute 'external_name' := 'F_VN_ExportContainer_String_GUID_D3BA1601_F2AB_D21E_B2A0_F8275CCD5A81'}
	(* Export the container elements into a string. Only possible for containers of type ContainerType_String_SINT. *)
	FUNCTION F_VN_ExportContainer_String : HRESULT
	VAR_INPUT
		ipContainer	:	ITcVnContainer;	(* Container of type ContainerType_String_SINT *)
	END_VAR
	VAR_IN_OUT CONSTANT
		sText	:	STRING;	(* Make sure to choose a sufficient STRING size! The required size can be determined using the function VnExportContainerSize. *)
	END_VAR
	VAR_INPUT
		nMaxLength	:	ULINT;	(* Maximum string length to export (including 0 termination). If the container content is longer, the string is cut off at nMaxLength - 1 and 0 termination is appended. In this case, S_FALSE is returned. *)
		hrPrev	:	HRESULT;	(* HRESULT indicating the result of previous operations (If SUCCEEDED(hrPrev) equals false, no operation is executed.) *)
	END_VAR

END_FUNCTION

// Functions/Basic Container Operations/F_VN_ExportSubContainer

	{attribute 'TcIecLibraryType'}
	{attribute 'external_name' := 'F_VN_ExportSubContainer_GUID_A4146C43_2410_DE91_A46D_AACA3959D213'}
	(* Export the container elements of a sub-container into a buffer (e.g. an array). Only possible for 2-dimensional containers with basic elements. *)
	FUNCTION F_VN_ExportSubContainer : HRESULT
	VAR_INPUT
		ipContainer	:	ITcVnContainer;	(* Container with basic elements *)
		nIndex	:	ULINT;	(* Index of the requested element *)
		pBuffer	:	PVOID;	(* Buffer to store the container elements (Make sure to allocate enough memory! The required size in bytes can be determined using the function F_VN_ExportSubContainerSize) *)
		nBufferSize	:	ULINT;	(* Size of the buffer memory in bytes *)
		hrPrev	:	HRESULT;	(* HRESULT indicating the result of previous operations (If SUCCEEDED(hrPrev) equals false, no operation is executed.) *)
	END_VAR

END_FUNCTION

// Functions/Basic Container Operations/F_VN_ExportSubContainerSize

	{attribute 'TcIecLibraryType'}
	{attribute 'external_name' := 'F_VN_ExportSubContainerSize_GUID_12553CB3_D785_D131_952B_25B69AEC0DA3'}
	(* Determine the required buffer size in bytes to store all container elements of a sub-container (number_of_Elements * size_per_Element). Only possible for 2-dimensional containers with basic elements. *)
	FUNCTION F_VN_ExportSubContainerSize : HRESULT
	VAR_INPUT
		ipContainer	:	ITcVnContainer;	(* Container with basic elements *)
		nIndex	:	ULINT;	(* Index of the requested element *)
	END_VAR
	VAR_IN_OUT
		nBufferSize	:	ULINT;	(* Output parameter containing the required buffer size *)
	END_VAR
	VAR_INPUT
		hrPrev	:	HRESULT;	(* HRESULT indicating the result of previous operations (If SUCCEEDED(hrPrev) equals false, no operation is executed.) *)
	END_VAR

END_FUNCTION

// Functions/Basic Container Operations/F_VN_ExportSubContainer_String

	{attribute 'TcIecLibraryType'}
	{attribute 'external_name' := 'F_VN_ExportSubContainer_String_GUID_C737E7C8_1EDD_DC02_967D_A4C415C31B3C'}
	(* Export the container elements of a sub-container into a string. Only possible for 2-dimensional containers of type ContainerType_Vector_String_SINT. *)
	FUNCTION F_VN_ExportSubContainer_String : HRESULT
	VAR_INPUT
		ipContainer	:	ITcVnContainer;	(* Container of type ContainerType_Vector_String_SINT *)
		nIndex	:	ULINT;	(* Index of the requested element *)
	END_VAR
	VAR_IN_OUT CONSTANT
		sText	:	STRING;	(* Make sure to choose a sufficient STRING size! The required size can be determined using the function VnExportSubContainerSize. *)
	END_VAR
	VAR_INPUT
		nMaxLength	:	ULINT;	(* Maximum string length to export (including 0 termination). If the container content is longer, the string is cut off at nMaxLength - 1 and 0 termination is appended. In this case, S_FALSE is returned. *)
		hrPrev	:	HRESULT;	(* HRESULT indicating the result of previous operations (If SUCCEEDED(hrPrev) equals false, no operation is executed.) *)
	END_VAR

END_FUNCTION

// Functions/Basic Container Operations/F_VN_ExtractContainerRange

	{attribute 'TcIecLibraryType'}
	{attribute 'external_name' := 'F_VN_ExtractContainerRange_GUID_C6D03928_E259_D8A9_B59F_D7B2EF67FCBB'}
	(* Copy the specified range of the source container into the destination container. (If the destination container already contains elements, they will be removed.) *)
	FUNCTION F_VN_ExtractContainerRange : HRESULT
	VAR_INPUT
		ipSrcContainer	:	ITcVnContainer;	(* Source container *)
		ipDestContainer	:	REFERENCE TO ITcVnContainer;	(* Destination container *)
		nFirstIdx	:	ULINT;	(* Index of the first element to copy *)
		nLastIdx	:	ULINT;	(* Index of the last element to copy *)
		hrPrev	:	HRESULT;	(* HRESULT indicating the result of previous operations (If SUCCEEDED(hrPrev) equals false, no operation is executed.) *)
	END_VAR

END_FUNCTION

// Functions/Basic Container Operations/F_VN_GetContainer

	{attribute 'TcIecLibraryType'}
	{attribute 'external_name' := 'F_VN_GetContainer_GUID_AF32E6AE_77A4_DD47_B39B_3296D865D110'}
	(* Gets a pointer to the current element converted into an ITcVnContainer interface and increment its reference counter (only possible for container types). (Alternatively use interface method .GetContainer.) *)
	FUNCTION F_VN_GetContainer : HRESULT
	VAR_INPUT
		ipIterator	:	ITcVnForwardIterator;	(* Iterator *)
		ipContainer	:	REFERENCE TO ITcVnContainer;	(* Returns the container interface *)
		hrPrev	:	HRESULT;	(* HRESULT indicating the result of previous operations (If SUCCEEDED(hrPrev) equals false, no operation is executed.) *)
	END_VAR

END_FUNCTION

// Functions/Basic Container Operations/F_VN_GetContainerExp

	{attribute 'TcIecLibraryType'}
	{attribute 'external_name' := 'F_VN_GetContainerExp_GUID_CB0E4C23_1A59_DDF9_995B_395B72C2A1F0'}
	(* Gets a pointer to the current element converted into an ITcVnContainer interface and increment its reference counter (only possible for container types). Additionally, an offset to increment or decrement the iterator afterwards can be provided. (expert function) *)
	FUNCTION F_VN_GetContainerExp : HRESULT
	VAR_INPUT
		ipIterator	:	ITcVnForwardIterator;	(* Iterator *)
		ipContainer	:	REFERENCE TO ITcVnContainer;	(* Returns the container interface *)
		nOffset	:	DINT;	(* Offset to increment (>0) or decrement (<0) the iterator afterwards *)
		hrPrev	:	HRESULT;	(* HRESULT indicating the result of previous operations (If SUCCEEDED(hrPrev) equals false, no operation is executed.) *)
	END_VAR

END_FUNCTION

// Functions/Basic Container Operations/F_VN_GetForwardIterator

	{attribute 'TcIecLibraryType'}
	{attribute 'external_name' := 'F_VN_GetForwardIterator_GUID_CB6532B0_BEBB_DB59_A007_0AD52C30B2B9'}
	(* Gets a forward iterator for the container. (Alternatively use interface method .GetForwardIterator.) *)
	FUNCTION F_VN_GetForwardIterator : HRESULT
	VAR_INPUT
		ipContainer	:	ITcVnContainer;	(* Container *)
		ipIterator	:	REFERENCE TO ITcVnForwardIterator;	(* Returns the iterator interface *)
		hrPrev	:	HRESULT;	(* HRESULT indicating the result of previous operations (If SUCCEEDED(hrPrev) equals false, no operation is executed.) *)
	END_VAR

END_FUNCTION

// Functions/Basic Container Operations/F_VN_GetNumberOfElements

	{attribute 'TcIecLibraryType'}
	{attribute 'external_name' := 'F_VN_GetNumberOfElements_GUID_490AF7C8_2253_DCE5_9300_885EF8D58FF2'}
	(* Gets the number of elements in the container. (Alternatively use interface method .getElementNum.) *)
	FUNCTION F_VN_GetNumberOfElements : HRESULT
	VAR_INPUT
		ipContainer	:	ITcVnContainer;	(* Container *)
	END_VAR
	VAR_IN_OUT
		nNumberOfElements	:	ULINT;	(* Returns the number of elements in ipContainer *)
	END_VAR
	VAR_INPUT
		hrPrev	:	HRESULT;	(* HRESULT indicating the result of previous operations (If SUCCEEDED(hrPrev) equals false, no operation is executed.) *)
	END_VAR

END_FUNCTION

// Functions/Basic Container Operations/F_VN_GetRandomAccessIterator

	{attribute 'TcIecLibraryType'}
	{attribute 'external_name' := 'F_VN_GetRandomAccessIterator_GUID_B7CB9E80_8EE2_D600_9681_946E9F837ABC'}
	(* Gets a random access iterator for the container. (Alternatively use interface method .GetRandomAccessIterator.) *)
	FUNCTION F_VN_GetRandomAccessIterator : HRESULT
	VAR_INPUT
		ipContainer	:	ITcVnContainer;	(* Container *)
		ipIterator	:	REFERENCE TO ITcVnRandomAccessIterator;	(* Returns the iterator interface *)
		hrPrev	:	HRESULT;	(* HRESULT indicating the result of previous operations (If SUCCEEDED(hrPrev) equals false, no operation is executed.) *)
	END_VAR

END_FUNCTION

// Functions/Basic Container Operations/F_VN_IncrementIterator

	{attribute 'TcIecLibraryType'}
	{attribute 'external_name' := 'F_VN_IncrementIterator_GUID_E1C3D766_B65F_D0A4_8686_2B95174E69BF'}
	(* Increment the iterator. (Alternatively use interface method .Increment.) *)
	FUNCTION F_VN_IncrementIterator : HRESULT
	VAR_INPUT
		ipIterator	:	ITcVnForwardIterator;	(* Iterator *)
		hrPrev	:	HRESULT;	(* HRESULT indicating the result of previous operations (If SUCCEEDED(hrPrev) equals false, no operation is executed.) *)
	END_VAR

END_FUNCTION

// Functions/Basic Container Operations/F_VN_IteratorDistance

	{attribute 'TcIecLibraryType'}
	{attribute 'external_name' := 'F_VN_IteratorDistance_GUID_547284EB_906F_D2FF_B98F_6F68610AA029'}
	(* Computes the distance between 2 iterators. *)
	FUNCTION F_VN_IteratorDistance : HRESULT
	VAR_INPUT
		ipIteratorFirst	:	ITcVnForwardIterator;	(* First iterator *)
		ipIteratorLast	:	ITcVnForwardIterator;	(* Last iterator *)
	END_VAR
	VAR_IN_OUT
		nDistance	:	LINT;	(* Returns the computed distance *)
	END_VAR
	VAR_INPUT
		hrPrev	:	HRESULT;	(* HRESULT indicating the result of previous operations (If SUCCEEDED(hrPrev) equals false, no operation is executed.) *)
	END_VAR

END_FUNCTION

// Functions/Basic Container Operations/F_VN_ReserveContainerMemory

	{attribute 'TcIecLibraryType'}
	{attribute 'external_name' := 'F_VN_ReserveContainerMemory_GUID_2EABDFD6_B39B_D33B_8B62_DDBC79AD0187'}
	(* Reserve container memory (call with maximum required number of elements before manually appending elements for better performance) *)
	FUNCTION F_VN_ReserveContainerMemory : HRESULT
	VAR_INPUT
		ipContainer	:	ITcVnContainer;	(* Container for which to reserve the memory *)
		nElements	:	ULINT;	(* Number of elements for which the container should reserve memory *)
		hrPrev	:	HRESULT;	(* HRESULT indicating the result of previous operations (If SUCCEEDED(hrPrev) equals false, no operation is executed.) *)
	END_VAR

END_FUNCTION

// Functions/Basic Container Operations/F_VN_ReverseContainer

	{attribute 'TcIecLibraryType'}
	{attribute 'external_name' := 'F_VN_ReverseContainer_GUID_BD93AF25_D177_DEAF_BD2B_50A1696DF709'}
	(* Reverse the container elements. *)
	FUNCTION F_VN_ReverseContainer : HRESULT
	VAR_INPUT
		ipContainer	:	ITcVnContainer;	(* Container to be reversed *)
		hrPrev	:	HRESULT;	(* HRESULT indicating the result of previous operations (If SUCCEEDED(hrPrev) equals false, no operation is executed.) *)
	END_VAR

END_FUNCTION

// Functions/Basic Container Operations/F_VN_SetContainer

	{attribute 'TcIecLibraryType'}
	{attribute 'external_name' := 'F_VN_SetContainer_GUID_6BF1C7E5_3C86_DC81_9F10_640B16B42809'}
	(* Sets the current element using an ITcVnContainer interface (only possible for container types). (Alternatively use interface method .SetContainer.) *)
	FUNCTION F_VN_SetContainer : HRESULT
	VAR_INPUT
		ipIterator	:	ITcVnForwardIterator;	(* Iterator *)
		ipContainer	:	ITcVnContainer;	(* Container interface of which the content is to be assigned to the current element *)
		hrPrev	:	HRESULT;	(* HRESULT indicating the result of previous operations (If SUCCEEDED(hrPrev) equals false, no operation is executed.) *)
	END_VAR

END_FUNCTION

// Functions/Basic Container Operations/F_VN_SetIteratorToBegin

	{attribute 'TcIecLibraryType'}
	{attribute 'external_name' := 'F_VN_SetIteratorToBegin_GUID_D9866549_071D_D0E9_AC92_8455ADFA36E1'}
	(* Sets the iterator to the first element of the container. (Alternatively use interface method .SetToBegin.) *)
	FUNCTION F_VN_SetIteratorToBegin : HRESULT
	VAR_INPUT
		ipIterator	:	ITcVnForwardIterator;	(* Iterator *)
		hrPrev	:	HRESULT;	(* HRESULT indicating the result of previous operations (If SUCCEEDED(hrPrev) equals false, no operation is executed.) *)
	END_VAR

END_FUNCTION

// Functions/Geometric and Coordinate Transformations/F_VN_AlignRotatedImageRegion

	{attribute 'TcIecLibraryType'}
	{attribute 'external_name' := 'F_VN_AlignRotatedImageRegion_GUID_B744E22A_57C4_D465_AFFE_4BFF6C38470B'}
	(* Copies the provided image region and aligns it to the image axes. *)
	FUNCTION F_VN_AlignRotatedImageRegion : HRESULT
	VAR_INPUT
		ipSrcImage	:	ITcVnImage;	(* Source image *)
		ipDestImage	:	REFERENCE TO ITcVnImage;	(* Destination image (An appropriate image will be created if required.) *)
	END_VAR
	VAR_IN_OUT
		stRegion	:	TcVnRotatedRectangle;	(* Image region to be aligned *)
	END_VAR
	VAR_INPUT
		hrPrev	:	HRESULT;	(* HRESULT indicating the result of previous operations (If SUCCEEDED(hrPrev) equals false, no operation is executed.) *)
	END_VAR

END_FUNCTION

// Functions/Geometric and Coordinate Transformations/F_VN_AlignRotatedImageRegionExp

	{attribute 'TcIecLibraryType'}
	{attribute 'external_name' := 'F_VN_AlignRotatedImageRegionExp_GUID_5B58E583_C806_D54E_86ED_358F67AF401B'}
	(* Copies the provided image region and aligns it to the image axes. (expert function) *)
	FUNCTION F_VN_AlignRotatedImageRegionExp : HRESULT
	VAR_INPUT
		ipSrcImage	:	ITcVnImage;	(* Source image *)
		ipDestImage	:	REFERENCE TO ITcVnImage;	(* Destination image (An appropriate image will be created if required.) *)
	END_VAR
	VAR_IN_OUT
		stRegion	:	TcVnRotatedRectangle;	(* Image region to be aligned *)
	END_VAR
	VAR_INPUT
		eInterpolationType	:	ETcVnInterpolationType;	(* Interpolation method *)
		eBorderInterpolation	:	ETcVnBorderInterpolationMethod;	(* Border interpolation method (ISOLATED not supported) *)
	END_VAR
	VAR_IN_OUT
		aBorderValue	:	TcVnVector4_LREAL;	(* Border value, if CONSTANT is used *)
	END_VAR
	VAR_INPUT
		hrPrev	:	HRESULT;	(* HRESULT indicating the result of previous operations (If SUCCEEDED(hrPrev) equals false, no operation is executed.) *)
	END_VAR

END_FUNCTION

// Functions/Geometric and Coordinate Transformations/F_VN_ApplyRotationToAffineTransformation

	{attribute 'TcIecLibraryType'}
	{attribute 'external_name' := 'F_VN_ApplyRotationToAffineTransformation_GUID_5AC8579C_2CD9_D86C_8FDB_A3CDAA357428'}
	(* Apply a rotation to an existing 2D affine transformation matrix. *)
	FUNCTION F_VN_ApplyRotationToAffineTransformation : HRESULT
	VAR_IN_OUT
		aTransformationMatrix	:	TcVnMatrix2x3_LREAL;	(* Affine transformation matrix to which the rotation is applied *)
	END_VAR
	VAR_INPUT
		fAngle	:	LREAL;	(* Angle in radians (positive means counter-clockwise) *)
		hrPrev	:	HRESULT;	(* HRESULT indicating the result of previous operations (If SUCCEEDED(hrPrev) equals false, no operation is executed.) *)
	END_VAR

END_FUNCTION

// Functions/Geometric and Coordinate Transformations/F_VN_ApplyRotationToAffineTransformationExp

	{attribute 'TcIecLibraryType'}
	{attribute 'external_name' := 'F_VN_ApplyRotationToAffineTransformationExp_GUID_81E3ACD3_6ADB_DA8F_9C5B_50CE3C95EE70'}
	(* Apply a rotation to an existing 2D affine transformation matrix. (expert function) *)
	FUNCTION F_VN_ApplyRotationToAffineTransformationExp : HRESULT
	VAR_IN_OUT
		aTransformationMatrix	:	TcVnMatrix2x3_LREAL;	(* Affine transformation matrix to which the rotation is applied *)
	END_VAR
	VAR_INPUT
		fAngle	:	LREAL;	(* Angle in radians (positive means counter-clockwise) *)
		bUsePreMultiplication	:	BOOL;	(* Select if pre- or post-multiplication should be used *)
		hrPrev	:	HRESULT;	(* HRESULT indicating the result of previous operations (If SUCCEEDED(hrPrev) equals false, no operation is executed.) *)
	END_VAR

END_FUNCTION

// Functions/Geometric and Coordinate Transformations/F_VN_ApplyScalingToAffineTransformation

	{attribute 'TcIecLibraryType'}
	{attribute 'external_name' := 'F_VN_ApplyScalingToAffineTransformation_GUID_82A1CAC1_E097_DD03_9F7E_2874CB4A972F'}
	(* Apply a scaling to an existing 2D affine transformation matrix. *)
	FUNCTION F_VN_ApplyScalingToAffineTransformation : HRESULT
	VAR_IN_OUT
		aTransformationMatrix	:	TcVnMatrix2x3_LREAL;	(* Affine transformation matrix to which the scaling is applied *)
	END_VAR
	VAR_INPUT
		fScaleX	:	LREAL;	(* Scaling factor in x direction *)
		fScaleY	:	LREAL;	(* Scaling factor in y direction *)
		hrPrev	:	HRESULT;	(* HRESULT indicating the result of previous operations (If SUCCEEDED(hrPrev) equals false, no operation is executed.) *)
	END_VAR

END_FUNCTION

// Functions/Geometric and Coordinate Transformations/F_VN_ApplyScalingToAffineTransformationExp

	{attribute 'TcIecLibraryType'}
	{attribute 'external_name' := 'F_VN_ApplyScalingToAffineTransformationExp_GUID_837F704E_8927_D653_A2AC_75E62E205C86'}
	(* Apply a scaling to an existing 2D affine transformation matrix. (expert function) *)
	FUNCTION F_VN_ApplyScalingToAffineTransformationExp : HRESULT
	VAR_IN_OUT
		aTransformationMatrix	:	TcVnMatrix2x3_LREAL;	(* Affine transformation matrix to which the scaling is applied *)
	END_VAR
	VAR_INPUT
		fScaleX	:	LREAL;	(* Scaling factor in x direction *)
		fScaleY	:	LREAL;	(* Scaling factor in y direction *)
		bUsePreMultiplication	:	BOOL;	(* Select if pre- or post-multiplication should be used *)
		hrPrev	:	HRESULT;	(* HRESULT indicating the result of previous operations (If SUCCEEDED(hrPrev) equals false, no operation is executed.) *)
	END_VAR

END_FUNCTION

// Functions/Geometric and Coordinate Transformations/F_VN_ApplyTranslationToAffineTransformation

	{attribute 'TcIecLibraryType'}
	{attribute 'external_name' := 'F_VN_ApplyTranslationToAffineTransformation_GUID_A4818B16_66FC_D373_9B81_85E30112E807'}
	(* Apply a translation to an existing 2D affine transformation matrix. *)
	FUNCTION F_VN_ApplyTranslationToAffineTransformation : HRESULT
	VAR_IN_OUT
		aTransformationMatrix	:	TcVnMatrix2x3_LREAL;	(* Affine transformation matrix to which the translation is applied *)
	END_VAR
	VAR_INPUT
		fDeltaX	:	LREAL;	(* Translation in x direction *)
		fDeltaY	:	LREAL;	(* Translation in y direction *)
		hrPrev	:	HRESULT;	(* HRESULT indicating the result of previous operations (If SUCCEEDED(hrPrev) equals false, no operation is executed.) *)
	END_VAR

END_FUNCTION

// Functions/Geometric and Coordinate Transformations/F_VN_ApplyTranslationToAffineTransformationExp

	{attribute 'TcIecLibraryType'}
	{attribute 'external_name' := 'F_VN_ApplyTranslationToAffineTransformationExp_GUID_3CECBEAC_167A_D85F_93D2_DDF27AB3C132'}
	(* Apply a translation to an existing 2D affine transformation matrix. (expert function) *)
	FUNCTION F_VN_ApplyTranslationToAffineTransformationExp : HRESULT
	VAR_IN_OUT
		aTransformationMatrix	:	TcVnMatrix2x3_LREAL;	(* Affine transformation matrix to which the translation is applied *)
	END_VAR
	VAR_INPUT
		fDeltaX	:	LREAL;	(* Translation in x direction *)
		fDeltaY	:	LREAL;	(* Translation in y direction *)
		bUsePreMultiplication	:	BOOL;	(* Select if pre- or post-multiplication should be used *)
		hrPrev	:	HRESULT;	(* HRESULT indicating the result of previous operations (If SUCCEEDED(hrPrev) equals false, no operation is executed.) *)
	END_VAR

END_FUNCTION

// Functions/Geometric and Coordinate Transformations/F_VN_ApplyYAxisInversionToAffineTransformation

	{attribute 'TcIecLibraryType'}
	{attribute 'external_name' := 'F_VN_ApplyYAxisInversionToAffineTransformation_GUID_23C504E2_E78F_DBED_ADAD_250401E827A8'}
	(* Apply an inversion of the y-axis direction to an existing 2D affine transformation matrix. *)
	FUNCTION F_VN_ApplyYAxisInversionToAffineTransformation : HRESULT
	VAR_IN_OUT
		aTransformationMatrix	:	TcVnMatrix2x3_LREAL;	(* Affine transformation matrix to which the inversion of the y-axis direction is applied *)
	END_VAR
	VAR_INPUT
		hrPrev	:	HRESULT;	(* HRESULT indicating the result of previous operations (If SUCCEEDED(hrPrev) equals false, no operation is executed.) *)
	END_VAR

END_FUNCTION

// Functions/Geometric and Coordinate Transformations/F_VN_ApplyYAxisInversionToAffineTransformationExp

	{attribute 'TcIecLibraryType'}
	{attribute 'external_name' := 'F_VN_ApplyYAxisInversionToAffineTransformationExp_GUID_8D7B884C_C66C_D607_8B97_D5C2EF0F83AF'}
	(* Apply an inversion of the y-axis direction to an existing 2D affine transformation matrix. (expert function) *)
	FUNCTION F_VN_ApplyYAxisInversionToAffineTransformationExp : HRESULT
	VAR_IN_OUT
		aTransformationMatrix	:	TcVnMatrix2x3_LREAL;	(* Affine transformation matrix to which the inversion of the y-axis direction is applied *)
	END_VAR
	VAR_INPUT
		bUsePreMultiplication	:	BOOL;	(* Select if pre- or post-multiplication should be used *)
		hrPrev	:	HRESULT;	(* HRESULT indicating the result of previous operations (If SUCCEEDED(hrPrev) equals false, no operation is executed.) *)
	END_VAR

END_FUNCTION

// Functions/Geometric and Coordinate Transformations/F_VN_ConvertCartesianToPolarAngleImage

	{attribute 'TcIecLibraryType'}
	{attribute 'external_name' := 'F_VN_ConvertCartesianToPolarAngleImage_GUID_9F88667D_1C68_D225_B40D_629BC5D284AF'}
	(* Converts cartesian coordinates (x, y) to polar angle. *)
	FUNCTION F_VN_ConvertCartesianToPolarAngleImage : HRESULT
	VAR_INPUT
		ipSrcImageX	:	ITcVnImage;	(* Source image containing the x values (elements of type REAL or LREAL) *)
		ipSrcImageY	:	ITcVnImage;	(* Source image containing the y values (Same element type as ipSrcImageX) *)
		ipDestImageAng	:	REFERENCE TO ITcVnImage;	(* Destination image containing the angles (Same element type as source images. An appropriate destination image will be created if required.) *)
		hrPrev	:	HRESULT;	(* HRESULT indicating the result of previous operations (If SUCCEEDED(hrPrev) equals false, no operation is executed.) *)
	END_VAR

END_FUNCTION

// Functions/Geometric and Coordinate Transformations/F_VN_ConvertCartesianToPolarAngleImageExp

	{attribute 'TcIecLibraryType'}
	{attribute 'external_name' := 'F_VN_ConvertCartesianToPolarAngleImageExp_GUID_950AC9BB_C3E5_D7F2_B055_44EF17B8A034'}
	(* Converts cartesian coordinates (x, y) to polar angle. (expert function) *)
	FUNCTION F_VN_ConvertCartesianToPolarAngleImageExp : HRESULT
	VAR_INPUT
		ipSrcImageX	:	ITcVnImage;	(* Source image containing the x values (elements of type REAL or LREAL) *)
		ipSrcImageY	:	ITcVnImage;	(* Source image containing the y values (Same element type as ipSrcImageX) *)
		ipDestImageAng	:	REFERENCE TO ITcVnImage;	(* Destination image containing the angles (Same element type as source images. An appropriate destination image will be created if required.) *)
		bAngleInDegrees	:	BOOL;	(* Specifys, if the angles should be in degrees or radians *)
		hrPrev	:	HRESULT;	(* HRESULT indicating the result of previous operations (If SUCCEEDED(hrPrev) equals false, no operation is executed.) *)
	END_VAR

END_FUNCTION

// Functions/Geometric and Coordinate Transformations/F_VN_ConvertCartesianToPolarAngles

	{attribute 'TcIecLibraryType'}
	{attribute 'external_name' := 'F_VN_ConvertCartesianToPolarAngles_GUID_6F76F677_FA20_D368_8CE7_8DDB1C4FB5F5'}
	(* Converts cartesian coordinates (x, y) to polar angle. *)
	FUNCTION F_VN_ConvertCartesianToPolarAngles : HRESULT
	VAR_INPUT
		ipSrcPointsCart	:	ITcVnContainer;	(* Container with cartesian points (ContainerType_Vector_TcVnPoint2_DINT or ContainerType_Vector_TcVnPoint2_REAL or ContainerType_Vector_TcVnPoint2_LREAL) *)
		ipDestAngles	:	REFERENCE TO ITcVnContainer;	(* Returns a container which is filled with the angles (ContainerType_Vector_REAL, if source points are of type TcVnPoint2_DINT or TcVnPoint2_REAL; else ContainerType_Vector_LREAL. Non-zero interface pointers are reused.) *)
		hrPrev	:	HRESULT;	(* HRESULT indicating the result of previous operations (If SUCCEEDED(hrPrev) equals false, no operation is executed.) *)
	END_VAR

END_FUNCTION

// Functions/Geometric and Coordinate Transformations/F_VN_ConvertCartesianToPolarAnglesExp

	{attribute 'TcIecLibraryType'}
	{attribute 'external_name' := 'F_VN_ConvertCartesianToPolarAnglesExp_GUID_D976057E_34F0_D46B_8F18_5DEA4C2D1490'}
	(* Converts cartesian coordinates (x, y) to polar angle. (expert function) *)
	FUNCTION F_VN_ConvertCartesianToPolarAnglesExp : HRESULT
	VAR_INPUT
		ipSrcPointsCart	:	ITcVnContainer;	(* Container with cartesian points (ContainerType_Vector_TcVnPoint2_DINT or ContainerType_Vector_TcVnPoint2_REAL or ContainerType_Vector_TcVnPoint2_LREAL) *)
		ipDestAngles	:	REFERENCE TO ITcVnContainer;	(* Returns a container which is filled with the angles (ContainerType_Vector_REAL, if source points are of type TcVnPoint2_DINT or TcVnPoint2_REAL; else ContainerType_Vector_LREAL. Non-zero interface pointers are reused.) *)
		bAngleInDegrees	:	BOOL;	(* Specify, if the angles should be in degrees or radians *)
		hrPrev	:	HRESULT;	(* HRESULT indicating the result of previous operations (If SUCCEEDED(hrPrev) equals false, no operation is executed.) *)
	END_VAR

END_FUNCTION

// Functions/Geometric and Coordinate Transformations/F_VN_ConvertCartesianToPolarImages

	{attribute 'TcIecLibraryType'}
	{attribute 'external_name' := 'F_VN_ConvertCartesianToPolarImages_GUID_70D8B5B2_5599_D52F_B3EB_3F2BEBBA1BAB'}
	(* Converts cartesian coordinates (x, y) to polar coordinates (magnitude, angle). *)
	FUNCTION F_VN_ConvertCartesianToPolarImages : HRESULT
	VAR_INPUT
		ipSrcImageX	:	ITcVnImage;	(* Source image containing the x values (elements of type REAL or LREAL) *)
		ipSrcImageY	:	ITcVnImage;	(* Source image containing the y values (Same element type as ipSrcImageX) *)
		ipDestImageMag	:	REFERENCE TO ITcVnImage;	(* Destination image containing the magnitudes (Same element type as source images. An appropriate destination image will be created if required.) *)
		ipDestImageAng	:	REFERENCE TO ITcVnImage;	(* Destination image containing the angles (Same element type as source images. An appropriate destination image will be created if required.) *)
		hrPrev	:	HRESULT;	(* HRESULT indicating the result of previous operations (If SUCCEEDED(hrPrev) equals false, no operation is executed.) *)
	END_VAR

END_FUNCTION

// Functions/Geometric and Coordinate Transformations/F_VN_ConvertCartesianToPolarImagesExp

	{attribute 'TcIecLibraryType'}
	{attribute 'external_name' := 'F_VN_ConvertCartesianToPolarImagesExp_GUID_4FA9D3EF_3EAD_D480_A4A3_F2BE14288262'}
	(* Converts cartesian coordinates (x, y) to polar coordinates (magnitude, angle). (expert function) *)
	FUNCTION F_VN_ConvertCartesianToPolarImagesExp : HRESULT
	VAR_INPUT
		ipSrcImageX	:	ITcVnImage;	(* Source image containing the x values (elements of type REAL or LREAL) *)
		ipSrcImageY	:	ITcVnImage;	(* Source image containing the y values (Same element type as ipSrcImageX) *)
		ipDestImageMag	:	REFERENCE TO ITcVnImage;	(* Destination image containing the magnitudes (Same element type as source images. An appropriate destination image will be created if required.) *)
		ipDestImageAng	:	REFERENCE TO ITcVnImage;	(* Destination image containing the angles (Same element type as source images. An appropriate destination image will be created if required.) *)
		bAngleInDegrees	:	BOOL;	(* Specifys, if the angles should be in degrees or radians *)
		hrPrev	:	HRESULT;	(* HRESULT indicating the result of previous operations (If SUCCEEDED(hrPrev) equals false, no operation is executed.) *)
	END_VAR

END_FUNCTION

// Functions/Geometric and Coordinate Transformations/F_VN_ConvertCartesianToPolarMagnitudeImage

	{attribute 'TcIecLibraryType'}
	{attribute 'external_name' := 'F_VN_ConvertCartesianToPolarMagnitudeImage_GUID_81E269ED_51E9_D46A_B3BC_3377C8758DD5'}
	(* Converts cartesian coordinates (x, y) to polar magnitude. *)
	FUNCTION F_VN_ConvertCartesianToPolarMagnitudeImage : HRESULT
	VAR_INPUT
		ipSrcImageX	:	ITcVnImage;	(* Source image containing the x values (elements of type REAL or LREAL) *)
		ipSrcImageY	:	ITcVnImage;	(* Source image containing the y values (Same element type as ipSrcImageX) *)
		ipDestImageMag	:	REFERENCE TO ITcVnImage;	(* Destination image containing the magnitudes (Same element type as source images. An appropriate destination image will be created if required.) *)
		hrPrev	:	HRESULT;	(* HRESULT indicating the result of previous operations (If SUCCEEDED(hrPrev) equals false, no operation is executed.) *)
	END_VAR

END_FUNCTION

// Functions/Geometric and Coordinate Transformations/F_VN_ConvertCartesianToPolarMagnitudes

	{attribute 'TcIecLibraryType'}
	{attribute 'external_name' := 'F_VN_ConvertCartesianToPolarMagnitudes_GUID_9F5AEA3F_A764_D98D_BD53_495A7BC718CB'}
	(* Converts cartesian coordinates (x, y) to polar magnitude. *)
	FUNCTION F_VN_ConvertCartesianToPolarMagnitudes : HRESULT
	VAR_INPUT
		ipSrcPointsCart	:	ITcVnContainer;	(* Container with cartesian points (ContainerType_Vector_TcVnPoint2_DINT or ContainerType_Vector_TcVnPoint2_REAL or ContainerType_Vector_TcVnPoint2_LREAL) *)
		ipDestMags	:	REFERENCE TO ITcVnContainer;	(* Returns a container which is filled with the magnitudes (ContainerType_Vector_REAL, if source points are of type TcVnPoint2_DINT or TcVnPoint2_REAL; else ContainerType_Vector_LREAL. Non-zero interface pointers are reused.) *)
		hrPrev	:	HRESULT;	(* HRESULT indicating the result of previous operations (If SUCCEEDED(hrPrev) equals false, no operation is executed.) *)
	END_VAR

END_FUNCTION

// Functions/Geometric and Coordinate Transformations/F_VN_ConvertCartesianToPolarPoints

	{attribute 'TcIecLibraryType'}
	{attribute 'external_name' := 'F_VN_ConvertCartesianToPolarPoints_GUID_931C5EAC_DA8F_D24B_855E_A63CC015AF6F'}
	(* Converts cartesian coordinates (x, y) to polar coordinates (magnitude, angle). *)
	FUNCTION F_VN_ConvertCartesianToPolarPoints : HRESULT
	VAR_INPUT
		ipSrcPointsCart	:	ITcVnContainer;	(* Container with cartesian points (ContainerType_Vector_TcVnPoint2_DINT or ContainerType_Vector_TcVnPoint2_REAL or ContainerType_Vector_TcVnPoint2_LREAL) *)
		ipDestPointsPolar	:	REFERENCE TO ITcVnContainer;	(* Returns a container which is filled with the converted points in polar coordinates (ContainerType_Vector_TcVnPoint2_REAL, if source points are of type TcVnPoint2_DINT or TcVnPoint2_REAL; else ContainerType_Vector_TcVnPoint2_LREAL. Non-zero interface pointers are reused.) *)
		hrPrev	:	HRESULT;	(* HRESULT indicating the result of previous operations (If SUCCEEDED(hrPrev) equals false, no operation is executed.) *)
	END_VAR

END_FUNCTION

// Functions/Geometric and Coordinate Transformations/F_VN_ConvertCartesianToPolarPointsExp

	{attribute 'TcIecLibraryType'}
	{attribute 'external_name' := 'F_VN_ConvertCartesianToPolarPointsExp_GUID_F3B3F847_BC39_DFD3_A48C_E996135FFD4E'}
	(* Converts cartesian coordinates (x, y) to polar coordinates (magnitude, angle). (expert function) *)
	FUNCTION F_VN_ConvertCartesianToPolarPointsExp : HRESULT
	VAR_INPUT
		ipSrcPointsCart	:	ITcVnContainer;	(* Container with cartesian points (ContainerType_Vector_TcVnPoint2_DINT or ContainerType_Vector_TcVnPoint2_REAL or ContainerType_Vector_TcVnPoint2_LREAL) *)
		ipDestPointsPolar	:	REFERENCE TO ITcVnContainer;	(* Returns a container which is filled with the converted points in polar coordinates (ContainerType_Vector_TcVnPoint2_REAL, if source points are of type TcVnPoint2_DINT or TcVnPoint2_REAL; else ContainerType_Vector_TcVnPoint2_LREAL. Non-zero interface pointers are reused.) *)
		bAngleInDegrees	:	BOOL;	(* Specifys, if the angles should be in degrees or radians *)
		hrPrev	:	HRESULT;	(* HRESULT indicating the result of previous operations (If SUCCEEDED(hrPrev) equals false, no operation is executed.) *)
	END_VAR

END_FUNCTION

// Functions/Geometric and Coordinate Transformations/F_VN_ConvertPolarToCartesianImages

	{attribute 'TcIecLibraryType'}
	{attribute 'external_name' := 'F_VN_ConvertPolarToCartesianImages_GUID_5DEF2919_1FD2_D1C7_AF63_EB577D058003'}
	(* Converts polar coordinates (magnitude, angle) to cartesian coordinates (x, y). *)
	FUNCTION F_VN_ConvertPolarToCartesianImages : HRESULT
	VAR_INPUT
		ipSrcImageMag	:	ITcVnImage;	(* Source image containing the magnitudes (elements of type REAL or LREAL) *)
		ipSrcImageAng	:	ITcVnImage;	(* Source image containing the angles (Same element type as ipSrcImageMag) *)
		ipDestImageX	:	REFERENCE TO ITcVnImage;	(* Destination image containing the x values (Same element type as source images. An appropriate destination image will be created if required.) *)
		ipDestImageY	:	REFERENCE TO ITcVnImage;	(* Destination image containing the y values (Same element type as source images. An appropriate destination image will be created if required.) *)
		hrPrev	:	HRESULT;	(* HRESULT indicating the result of previous operations (If SUCCEEDED(hrPrev) equals false, no operation is executed.) *)
	END_VAR

END_FUNCTION

// Functions/Geometric and Coordinate Transformations/F_VN_ConvertPolarToCartesianImagesExp

	{attribute 'TcIecLibraryType'}
	{attribute 'external_name' := 'F_VN_ConvertPolarToCartesianImagesExp_GUID_02B87E65_AD5C_DAF8_9D05_58102819EF4E'}
	(* Converts polar coordinates (magnitude, angle) to cartesian coordinates (x, y). (expert function) *)
	FUNCTION F_VN_ConvertPolarToCartesianImagesExp : HRESULT
	VAR_INPUT
		ipSrcImageMag	:	ITcVnImage;	(* Source image containing the magnitudes (elements of type REAL or LREAL) *)
		ipSrcImageAng	:	ITcVnImage;	(* Source image containing the angles (Same element type as ipSrcImageMag) *)
		ipDestImageX	:	REFERENCE TO ITcVnImage;	(* Destination image containing the x values (Same element type as source images. An appropriate destination image will be created if required.) *)
		ipDestImageY	:	REFERENCE TO ITcVnImage;	(* Destination image containing the y values (Same element type as source images. An appropriate destination image will be created if required.) *)
		bAngleInDegrees	:	BOOL;	(* Specifys, if the angles are in degrees or radians *)
		hrPrev	:	HRESULT;	(* HRESULT indicating the result of previous operations (If SUCCEEDED(hrPrev) equals false, no operation is executed.) *)
	END_VAR

END_FUNCTION

// Functions/Geometric and Coordinate Transformations/F_VN_ConvertPolarToCartesianPoints

	{attribute 'TcIecLibraryType'}
	{attribute 'external_name' := 'F_VN_ConvertPolarToCartesianPoints_GUID_D594A63C_24AA_DB8A_983B_AE78C4FCB253'}
	(* Converts polar coordinates (magnitude, angle) to cartesian coordinates (x, y). *)
	FUNCTION F_VN_ConvertPolarToCartesianPoints : HRESULT
	VAR_INPUT
		ipSrcPointsPolar	:	ITcVnContainer;	(* Container with polar coordinates (ContainerType_Vector_TcVnPoint2_REAL or ContainerType_Vector_TcVnPoint2_LREAL) *)
		ipDestPointsCart	:	REFERENCE TO ITcVnContainer;	(* Returns a container which is filled with the converted points in cartesian coordinates (same type ID as ipSrcPointsPolar. Non-zero interface pointers are reused.) *)
		hrPrev	:	HRESULT;	(* HRESULT indicating the result of previous operations (If SUCCEEDED(hrPrev) equals false, no operation is executed.) *)
	END_VAR

END_FUNCTION

// Functions/Geometric and Coordinate Transformations/F_VN_ConvertPolarToCartesianPointsExp

	{attribute 'TcIecLibraryType'}
	{attribute 'external_name' := 'F_VN_ConvertPolarToCartesianPointsExp_GUID_8982F90B_1EC9_DAB7_92CC_22CDBD07B99A'}
	(* Converts polar coordinates (magnitude, angle) to cartesian coordinates (x, y). (expert function) *)
	FUNCTION F_VN_ConvertPolarToCartesianPointsExp : HRESULT
	VAR_INPUT
		ipSrcPointsPolar	:	ITcVnContainer;	(* Container with polar coordinates (ContainerType_Vector_TcVnPoint2_REAL or ContainerType_Vector_TcVnPoint2_LREAL) *)
		ipDestPointsCart	:	REFERENCE TO ITcVnContainer;	(* Returns a container which is filled with the converted points in cartesian coordinates (same type ID as ipSrcPointsPolar. Non-zero interface pointers are reused.) *)
		bAngleInDegrees	:	BOOL;	(* Specifys, if the angles are in degrees or radians *)
		hrPrev	:	HRESULT;	(* HRESULT indicating the result of previous operations (If SUCCEEDED(hrPrev) equals false, no operation is executed.) *)
	END_VAR

END_FUNCTION

// Functions/Geometric and Coordinate Transformations/F_VN_DecomposeAffineTransformation

	{attribute 'TcIecLibraryType'}
	{attribute 'external_name' := 'F_VN_DecomposeAffineTransformation_GUID_80D87A6F_1825_D43E_987D_6360D44517E8'}
	(* Decompose an affine transformation matrix and return the rotation angle (clockwise) in radian. The decomposition method assumes the following order of transformation: Translation, Rotation, Scale, and Skew. *)
	FUNCTION F_VN_DecomposeAffineTransformation : HRESULT
	VAR_IN_OUT
		aAffineTransform	:	TcVnMatrix2x3_LREAL;	(* Affine transformation matrix *)
		fRotationAngle	:	LREAL;	(* Rotation angle (radian) in the clockwise direction. The rotation center is the origin point (0,0) *)
	END_VAR
	VAR_INPUT
		hrPrev	:	HRESULT;	(* HRESULT indicating the result of previous operations (If SUCCEEDED(hrPrev) equals false, no operation is executed.) *)
	END_VAR

END_FUNCTION

// Functions/Geometric and Coordinate Transformations/F_VN_DecomposeAffineTransformationExp

	{attribute 'TcIecLibraryType'}
	{attribute 'external_name' := 'F_VN_DecomposeAffineTransformationExp_GUID_827B06F3_0120_D8BD_B5FE_B035E009A279'}
	(* Decompose an affine transformation matrix and return the rotation angle (clockwise) in radian, translation vector (pixels), scale, and skew vectors (angle in radian). The decomposition method assumes the following order of transformation: Translation, Rotation, Scale, and Skew. *)
	FUNCTION F_VN_DecomposeAffineTransformationExp : HRESULT
	VAR_IN_OUT
		aAffineTransform	:	TcVnMatrix2x3_LREAL;	(* Affine transformation matrix *)
		fRotationAngle	:	LREAL;	(* Rotation angle (radian) in the clockwise direction. The rotation center is the origin point (0,0) *)
		aTranslationVector	:	TcVnVector2_LREAL;	(* 2D translation vector. The values are in pixels *)
		aScaleVector	:	TcVnVector2_LREAL;	(* 2D scale vector  *)
		aSkewVector	:	TcVnVector2_LREAL;	(* 2D skew vector. The values are the skew angles in x and y directions in radian *)
	END_VAR
	VAR_INPUT
		hrPrev	:	HRESULT;	(* HRESULT indicating the result of previous operations (If SUCCEEDED(hrPrev) equals false, no operation is executed.) *)
	END_VAR

END_FUNCTION

// Functions/Geometric and Coordinate Transformations/F_VN_DecomposeHomography

	{attribute 'TcIecLibraryType'}
	{attribute 'external_name' := 'F_VN_DecomposeHomography_GUID_80FDA367_8345_D846_B639_15ECC43470CB'}
	(* Decompose a homography matrix into four solutions of rotation, translation, and plane normal. It returns two solutions (Ra, Ta, Nb) and (Rb, Tb, Nb). The third and the fourth solutions can be calculated as follows: (Ra, -Ta, -Na) and (Rb, -Tb, -Nb). *)
	FUNCTION F_VN_DecomposeHomography : HRESULT
	VAR_IN_OUT
		aHomography	:	TcVnMatrix3x3_LREAL;	(* Homography matrix (a perspective transformation between two planes) *)
		aCameraMatrix	:	TcVnMatrix3x3_LREAL;	(* Camera matrix *)
		aRotationMatrixA	:	TcVnMatrix3x3_LREAL;	(* Rotation matrix of the first solution (Ra) *)
		aTranslationVectorA	:	TcVnVector3_LREAL;	(* Translation vector of the first solution (Ta) *)
		aNormVectorA	:	TcVnVector3_LREAL;	(* Norm vector of the first solution (Na) *)
		aRotationMatrixB	:	TcVnMatrix3x3_LREAL;	(* Rotation matrix of the second solution (Rb) *)
		aTranslationVectorB	:	TcVnVector3_LREAL;	(* Translation vector of the second solution (Tb) *)
		aNormVectorB	:	TcVnVector3_LREAL;	(* Norm vector of the second solution Nb *)
	END_VAR
	VAR_INPUT
		hrPrev	:	HRESULT;	(* HRESULT indicating the result of previous operations (If SUCCEEDED(hrPrev) equals false, no operation is executed.) *)
	END_VAR
	VAR_OUTPUT
		nSolutions	:	UDINT;	(* Returns the number of solutions. In normal cases, it is equal four.  *)
	END_VAR

END_FUNCTION

// Functions/Geometric and Coordinate Transformations/F_VN_DecomposeHomographyExp

	{attribute 'TcIecLibraryType'}
	{attribute 'external_name' := 'F_VN_DecomposeHomographyExp_GUID_FC5EFEAF_6F1D_D442_B76D_F6368456E965'}
	(* Decompose a homography matrix and verify four solutions of rotation, translation, and plane normal. It uses visible reference points being in front of the camera to confirm which solution(s) of the four solutions (maximum two solutions) are consistent with all reference points. *)
	FUNCTION F_VN_DecomposeHomographyExp : HRESULT
	VAR_IN_OUT
		aHomography	:	TcVnMatrix3x3_LREAL;	(* Homography matrix (a perspective transformation between two planes) *)
		aCameraMatrix	:	TcVnMatrix3x3_LREAL;	(* Camera matrix *)
		aRotationMatrixA	:	TcVnMatrix3x3_LREAL;	(* Rotation matrix of the first solution (Ra) *)
		aTranslationVectorA	:	TcVnVector3_LREAL;	(* Translation vector of the first solution (Ta) *)
		aNormVectorA	:	TcVnVector3_LREAL;	(* Norm vector of the first solution (Na) *)
		aRotationMatrixB	:	TcVnMatrix3x3_LREAL;	(* Rotation matrix of the second solution (Rb) *)
		aTranslationVectorB	:	TcVnVector3_LREAL;	(* Translation vector of the second solution (Tb) *)
		aNormVectorB	:	TcVnVector3_LREAL;	(* Norm vector of the second solution (Nb) *)
	END_VAR
	VAR_INPUT
		ipPointsSrc	:	ITcVnContainer;	(* Container with source points (ContainerType_Vector_TcVnPoint2_REAL) *)
		ipPointsDes	:	ITcVnContainer;	(* Container with destination points (same number as ipPoints1, ContainerType_Vector_TcVnPoint2_REAL) *)
		ipInlierMask	:	ITcVnContainer;	(* A mask marking the inliers (optional, set to 0 if not available; ContainerType_Vector_SINT or ContainerType_Vector_USINT) *)
		hrPrev	:	HRESULT;	(* HRESULT indicating the result of previous operations (If SUCCEEDED(hrPrev) equals false, no operation is executed.) *)
	END_VAR
	VAR_OUTPUT
		nSolutions	:	UDINT;	(* Return the number of true potential solutions [0,1, or 2].
							0: no true potential solutions for the given corresponding points are confirmed.
							1: the solution (Ra, Ta, Na) is confirmed.
							2: both solution (Ra, Ta, Na) and (Rb, Tb, Nb) are confirmed.
							In all cases the function returns two solutions (Ra, Ta, Nb) and (Rb, Tb, Nb). The third and the fourth solutions can be calculated as follows: (Ra, -Ta, -Na) and (Rb, -Tb, -Nb).
						 *)
	END_VAR

END_FUNCTION

// Functions/Geometric and Coordinate Transformations/F_VN_FlipImage

	{attribute 'TcIecLibraryType'}
	{attribute 'external_name' := 'F_VN_FlipImage_GUID_50BE975F_F837_DC78_B6F2_3204DBCC1FCC'}
	(* Flip an image (mirror and shift back to prior coordinates). *)
	FUNCTION F_VN_FlipImage : HRESULT
	VAR_INPUT
		ipSrcImage	:	ITcVnImage;	(* Source image *)
		ipDestImage	:	REFERENCE TO ITcVnImage;	(* Destination image (An appropriate destination image will be created if required.) *)
		eFlipAxis	:	ETcVnFlipAxis;	(* Selects the axis around which to flip the image *)
		hrPrev	:	HRESULT;	(* HRESULT indicating the result of previous operations (If SUCCEEDED(hrPrev) equals false, no operation is executed.) *)
	END_VAR

END_FUNCTION

// Functions/Geometric and Coordinate Transformations/F_VN_GenerateAffineTransformationUnitMatrix2D

	{attribute 'TcIecLibraryType'}
	{attribute 'external_name' := 'F_VN_GenerateAffineTransformationUnitMatrix2D_GUID_167BD96A_DB2B_D249_B184_A39F0926B1D6'}
	(* Generate an affine transformation 2D unit matrix. *)
	FUNCTION F_VN_GenerateAffineTransformationUnitMatrix2D : HRESULT
	VAR_IN_OUT
		aTransformationMatrix	:	TcVnMatrix2x3_LREAL;	(* Resulting affine transformation unit matrix *)
	END_VAR
	VAR_INPUT
		hrPrev	:	HRESULT;	(* HRESULT indicating the result of previous operations (If SUCCEEDED(hrPrev) equals false, no operation is executed.) *)
	END_VAR

END_FUNCTION

// Functions/Geometric and Coordinate Transformations/F_VN_GetAffineTransformation

	{attribute 'TcIecLibraryType'}
	{attribute 'external_name' := 'F_VN_GetAffineTransformation_GUID_6799CC81_5E3E_D6E6_B5F5_0981AA79AD7A'}
	(* Calculate the affine transformation between three corresponding point pairs. The points mark the corners of the corresponding triangles. *)
	FUNCTION F_VN_GetAffineTransformation : HRESULT
	VAR_IN_OUT
		aSrcPoints	:	TcVnArray3_Point2_REAL;	(* Source points *)
		aDestPoints	:	TcVnArray3_Point2_REAL;	(* Destination points *)
		aTransformationMatrix	:	TcVnMatrix2x3_LREAL;	(* Resulting transformation matrix *)
	END_VAR
	VAR_INPUT
		hrPrev	:	HRESULT;	(* HRESULT indicating the result of previous operations (If SUCCEEDED(hrPrev) equals false, no operation is executed.) *)
	END_VAR

END_FUNCTION

// Functions/Geometric and Coordinate Transformations/F_VN_GetAffineTransformation2D

